// TwinCAT 3 PLC project TcoUrRobotics
// Title: TcoUrRobotics
// Company: Vortex.Library
// Author: TcOpenGroup
// ProjectVersion: 0.6.0.913
// ProgramVersion: 3.1.4024.12
// libraries:
//   Tc2_Standard, * (Beckhoff Automation GmbH)
//   Tc2_System, * (Beckhoff Automation GmbH)
//   Tc2_Utilities, * (Beckhoff Automation GmbH)
//   Tc3_Module, * (Beckhoff Automation GmbH)
//   TcoAbstractions, 0.6.0.913 (Vortex.Library)
//   TcoCore, 0.6.0.913 (Vortex.Library)
//   TcoIo, 0.6.0.913 (Vortex.Library)
//   TcoUtilities, 0.6.0.913 (Vortex.Library)
// project tree:
//   DUTs/ eTcoUrRoboticsRobotMode.TcDUT, TcoUrRoboticsInputData.TcDUT, TcoUrRoboticsOutputData.TcDUT, TcoUrRobotics_Config_v_1_x_x.TcDUT, TcoUrRobotics_Control_v_1_x_x.TcDUT, TcoUrRobotics_State_v_1_x_x.TcDUT, TcoUrRobotics_Status_v_1_x_x.TcDUT
//   DUTs/Input/ TcoUrRoboticsT2OBitRegs.TcDUT, TcoUrRoboticsT2OFloatRegs.TcDUT, TcoUrRoboticsT2ORobot.TcDUT, TcoUrRoboticsT2OIntRegs.TcDUT, TcoUrRoboticsT2OIo.TcDUT, TcoUrRoboticsT2OJoints.TcDUT, TcoUrRoboticsT2OSafety.TcDUT, TcoUrRoboticsT2OTcp.TcDUT, TcoUrRoboticsT2OTool.TcDUT
//   DUTs/Out/ TcoUrRobotics_O2TIo.TcDUT, TcoUrRobotics_O2TReg.TcDUT, TcoUrRobotics_O2TRobot.TcDUT
//   / PlcTask.TcTTO
//   POUs/ GetRobotModeDescription.TcPOU, MAIN.TcPOU
//   POUs/Prototypes/Cb3/IO/ TcoUrCb3_Inputs_v_3_x_x.TcDUT, TcoUrCb3_IO_v_3_x_x.TcDUT, TcoUrCb3_Outputs_v_3_x_x.TcDUT
//   POUs/Prototypes/Cb3/ TcoUrCb3_v_3_x_x.TcPOU
//   POUs/Prototypes/Eseries/IO/ TcoUrEseries_Inputs_v_5_x_x.TcDUT, TcoUrEseries_IO_v_5_x_x.TcDUT, TcoUrEseries_Outputs_v_5_x_x.TcDUT
//   POUs/Prototypes/Eseries/ TcoUrEseries_v_5_x_x.TcPOU
//   POUs/Prototypes/Generic/Inputs/ TcoUrRobotics_T2O_State_IO.TcDUT, TcoUrRobotics_T2O_IO_IO.TcDUT, TcoUrRobotics_T2O_Joints_IO.TcDUT, TcoUrRobotics_T2O_TCP_IO.TcDUT, TcoUrRobotics_T2O_BitRegs_IO.TcDUT, TcoUrRobotics_T2O_IntRegs_IO.TcDUT, TcoUrRobotics_T2O_FloatRegs_IO.TcDUT
//   POUs/Prototypes/Generic/Outputs/ TcoUrRobotics_O2T_Reg1_IO.TcDUT, TcoUrRobotics_O2T_Reg2_IO.TcDUT, TcoUrRobotics_O2T_Robot_IO.TcDUT
//   POUs/Prototypes/RoboticsTasks/Starts/ StartAtMainTask.TcPOU, StartMotorsAndProgramTask.TcPOU, StartMotorsProgramAndMovementsTask.TcPOU, StartMotorsTask.TcPOU, StartMovementsTask.TcPOU, StartProgramTask.TcPOU
//   POUs/Prototypes/RoboticsTasks/Stops/ StopMovementsAndProgramTask.TcPOU, StopMovementsTask.TcPOU, StopProgramTask.TcPOU
//   POUs/Prototypes/RoboticsTasks/ TcoUrRoboticsTask.TcPOU
// real-time tasks:
//   TASK PlcTask: cycle T#10ms, priority 20, ADS port 350
//   TASK PlcTask1: cycle T#10ms, priority 1, ADS port 351
//   TASK PN: cycle T#32ms, priority 2, ADS port 301
// I/O:
//   DEVICE Device 4 (EtherCAT) (disabled), AmsNetId 172.20.10.104.5.1
//     Term 1 (EK1100) [EK1100 EtherCAT Coupler (2A E-Bus)]
//       Term 2 (EL1008) [EL1008 8Ch. Dig. Input 24V, 3ms]
//       Term 3 (EL2008) [EL2008 8Ch. Dig. Output 24V, 0.5A]
//       Term 4 (EL3052) [EL3052 2Ch. Ana. Input 4-20mA]
//       Term 5 (EL9576) [EL9576 Brake chopper terminal]
//       Term 6 (EL7211-0010) [EL7211-0010 1Ch. MDP742 Servo motor output stage with OCT (50V, 4.5A RMS)]
//       Term 14 (EL7047) [EL7047 1Ch. Stepper motor output stage (50V, 5A)]
//       Term 8 (EL9011) [EL9011 End Terminal]
//   DEVICE Device 1 (EtherCAT) (disabled), AmsNetId 192.168.4.1.2.1
//     Drive 7 (IndraDrive MPB20) [IndraDrive MPB20]
//   DEVICE Device 2 (EtherCAT) (disabled), AmsNetId 192.168.4.1.3.1
//     Term 1 (EK1200) [EK1200-5000 EtherCAT Power supply (2A E-Bus)]
//       Term 10 (EK1122) [EK1122 2 port EtherCAT junction]
//       Term 13 (EL6631) [EL6631 PROFINET IO Controller]
//       Term 12 (EL1809) [EL1809 16Ch. Dig. Input 24V, 3ms]
//       Term 13 (EL2809) [EL2809 16Ch. Dig. Output 24V, 0.5A]
//       Term 15 (EL4004) [EL4004 4Ch. Ana. Output 0-10V, 12bit]
//       Term 16 (EL7342) [EL7342 2Ch. DC motor output stage (50V, 3.5A)]
//       Term 17 (EL4004) [EL4004 4Ch. Ana. Output 0-10V, 12bit]
//       Term 18 (EL6001) [EL6001 Interface (RS232)]
//       Term 10 (EL9011) [EL9011 End Terminal]
//   DEVICE Device 5 (Profinet Controller) (disabled), AmsNetId 192.168.4.1.6.1
//     ur-op-80r [Universal Robots A/S UR IO device, for PNIO controller with PDev 0000201]
//       modules: Term 1 (DAP Module), Term 3 (1_T2O State), Term 4 (2_T2O IO), Term 5 (3_T2O Joints), Term 6 (4_T2O TCP), Term 7 (5_T2O General Purpose Bit Registers), Term 8 (6_T2O General Purpose Int Registers), Term 9 (7_T2O General Purpose Float Registers), Term 10 (8_O2T Robot IO), Term 11 (9_O2T General Purpose Registers 1), Term 12 (10_O2T General Purpose Registers 2)
// variable links:
//   TcoUrRoboticsTests/TcoUrRoboticsTests Instance <-> Device 2 (EtherCAT)/Term 1 (EK1200)/Term 13 (EL2809)
//     PlcTask1 Outputs/GVL.A2[0] <-> Channel 1/Output
//     PlcTask1 Outputs/GVL.A2[1] <-> Channel 2/Output
//   TcoUrRoboticsTests/TcoUrRoboticsTests Instance <-> Device 5 (Profinet Controller)/ur-op-80r
//     PlcTask1 Inputs/GVL.Robot1.In.BitRegs.bArray <-> API/Term 7 (5_T2O General Purpose Bit Registers)/Subterm 9 (5_T2O General Purpose Bit Registers)/Inputs/T2O Bit Registers
//     PlcTask1 Inputs/GVL.Robot1.In.FloatRegs.bArray <-> API/Term 9 (7_T2O General Purpose Float Registers)/Subterm 11 (7_T2O General Purpose Float Registers)/Inputs/T2O Float Registers
//     PlcTask1 Inputs/GVL.Robot1.In.IO.bArray <-> API/Term 4 (2_T2O IO)/Subterm 6 (2_T2O IO)/Inputs/T2O IO
//     PlcTask1 Inputs/GVL.Robot1.In.IntRegs.bArray <-> API/Term 8 (6_T2O General Purpose Int Registers)/Subterm 10 (6_T2O General Purpose Int Registers)/Inputs/T2O Int Registers
//     PlcTask1 Inputs/GVL.Robot1.In.Joints.bArray <-> API/Term 5 (3_T2O Joints)/Subterm 7 (3_T2O Joints)/Inputs/T2O Joints
//     PlcTask1 Inputs/GVL.Robot1.In.State.bArray <-> API/Term 3 (1_T2O State)/Subterm 5 (1_T2O State)/Inputs/T2O State
//     PlcTask1 Inputs/GVL.Robot1.In.TCP.bArray <-> API/Term 6 (4_T2O TCP)/Subterm 8 (4_T2O TCP)/Inputs/T2O TCP
//     PlcTask1 Inputs/GVL.Robot1.PnIoBoxDiag <-> Inputs/PnIoBoxDiag
//     PlcTask1 Inputs/GVL.Robot1.PnIoBoxState <-> Inputs/PnIoBoxState
//     PlcTask1 Outputs/GVL.Robot1.Out.Reg1.bArray <-> API/Term 11 (9_O2T General Purpose Registers 1)/Subterm 13 (9_O2T General Purpose Registers 1)/Outputs/O2T Reg 1
//     PlcTask1 Outputs/GVL.Robot1.Out.Reg2.bArray <-> API/Term 12 (10_O2T General Purpose Registers 2)/Subterm 14 (10_O2T General Purpose Registers 2)/Outputs/O2T Reg 2
//     PlcTask1 Outputs/GVL.Robot1.Out.RobotIO.bArray <-> API/Term 10 (8_O2T Robot IO)/Subterm 12 (8_O2T Robot IO)/Outputs/O2T IO

CONFIGURATION TcoUrRobotics
    RESOURCE PLC ON TwinCAT3
        TASK PlcTask(INTERVAL := T#10ms, PRIORITY := 20);
        PROGRAM MAIN WITH PlcTask : MAIN;
    END_RESOURCE
END_CONFIGURATION

// ---- DUTs/eTcoUrRoboticsRobotMode.TcDUT
{attribute 'qualified_only'}
{attribute 'strict'}
TYPE eTcoUrRoboticsRobotMode :
(
    DISCONNECTED := 0,
    SAFETY := 1,
    BOOTING := 2,
    POWER_OFF := 3,
    POWER_ON := 4,
    IDLE := 5,
    BACKDRIVE := 6,
    RUNNING := 7,
    UPDATING_FIRMWARE := 8
);
END_TYPE

// ---- DUTs/Input/TcoUrRoboticsT2OBitRegs.TcDUT
TYPE TcoUrRoboticsT2OBitRegs :
STRUCT
    {attribute addProperty Name "<#Bit registers#>"}
    Register : ARRAY[0..63] OF BOOL;
END_STRUCT
END_TYPE

// ---- DUTs/Input/TcoUrRoboticsT2OFloatRegs.TcDUT
TYPE TcoUrRoboticsT2OFloatRegs :
STRUCT
    {attribute addProperty Name "<#Float registers#>"}
    Register : ARRAY[0..23] OF REAL;
END_STRUCT
END_TYPE

// ---- DUTs/Input/TcoUrRoboticsT2ORobot.TcDUT
TYPE TcoUrRoboticsT2ORobot :
STRUCT
    {attribute addProperty Name "<#Controller major version#>"}
    ControllerMajorVersion : USINT;
    {attribute addProperty Name "<#Controller minor version#>"}
    ControllerMinorVersion : USINT;
    {attribute addProperty Name "<#Reserved#>"}
    Reserved : UINT;
    {attribute addProperty Name "<#Robot mode#>"}
    RobotMode : USINT;
    {attribute addProperty Name "<#Real time machine seconds#>"}
    RealtimeMachineSeconds : USINT;
    {attribute addProperty Name "<#Real time machine milliseconds#>"}
    RealtimeMachineMilliseconds : UINT;
    {attribute addProperty Name "<#Real time machine minutes#>"}
    RealtimeMachineMinutes : USINT;
    {attribute addProperty Name "<#Real time machine hours#>"}
    RealtimeMachineHours : USINT;
    {attribute addProperty Name "<#Real time machine days#>"}
    RealtimeMachineDays : UINT;
    {attribute addProperty Name "<#Robot current [A]#>"}
    RobotCurrent : REAL;
    {attribute addProperty Name "<#PW: Is power on#>"}
    PW_IsPowerOn : BOOL;
    {attribute addProperty Name "<#PR: Is program running#>"}
    PR_IsProgramRunning : BOOL;
    {attribute addProperty Name "<#TB: Is teach button pressed#>"}
    TB_IsTeachButtonPressed : BOOL;
    {attribute addProperty Name "<#PB: Is power button pressed#>"}
    PB_IsPowerButtonPressed : BOOL;
    {attribute addProperty Name "<#Speed slider fraction#>"}
    SpeedSliderFraction : REAL;
END_STRUCT
END_TYPE

// ---- DUTs/Input/TcoUrRoboticsT2OIntRegs.TcDUT
TYPE TcoUrRoboticsT2OIntRegs :
STRUCT
    {attribute addProperty Name "<#Int registers#>"}
    Register : ARRAY[0..23] OF DINT;
END_STRUCT
END_TYPE

// ---- DUTs/Input/TcoUrRoboticsT2OIo.TcDUT
TYPE TcoUrRoboticsT2OIo :
STRUCT
    {attribute addProperty Name "<#Standard digital inputs#>"}
    StandardDigitalInputs : USINT;
    {attribute addProperty Name "<#Configurable digital inputs#>"}
    ConfigurableDigitalInputs : USINT;
    {attribute addProperty Name "<#Standard digital outputs#>"}
    StandardDigitalOutputs : USINT;
    {attribute addProperty Name "<#Configurable digital outputs#>"}
    ConfigurableDigitalOutputs : USINT;
    {attribute addProperty Name "<#Analog I/O types#>"}
    AnalogIoTypes : USINT;
    {attribute addProperty Name "<#Standard analog input [A or V]#>"}
    StandardAnalogInput : ARRAY[0..1] OF REAL;
    {attribute addProperty Name "<#Standard analog output [A or V]#>"}
    StandardAnalogOutput : ARRAY[0..1] OF REAL;
    {attribute addProperty Name "<#I/O current [A]#>"}
    Current : REAL;
    {attribute addProperty Name "<#Euromap67 input bits#>"}
    Euromap67InputBits : ARRAY[0..31] OF BOOL;
    {attribute addProperty Name "<#Euromap67 output bits#>"}
    Euromap67OutputBits : ARRAY[0..31] OF BOOL;
    {attribute addProperty Name "<#Euromap67 24V voltage#>"}
    Euromap6724Voltage : REAL;
    {attribute addProperty Name "<#Euromap67 24V current#>"}
    Euromap6724VCurrent : REAL;
END_STRUCT
END_TYPE

// ---- DUTs/Input/TcoUrRoboticsT2OJoints.TcDUT
TYPE TcoUrRoboticsT2OJoints :
STRUCT
    {attribute addProperty Name "<#Joint position [rad]#>"}
    JointPosition : ARRAY[0..5] OF REAL;
    {attribute addProperty Name "<#Joint velocity [rad/s]#>"}
    JointVelocity : ARRAY[0..5] OF REAL;
    {attribute addProperty Name "<#Joint current [A]#>"}
    JointCurrent : ARRAY[0..5] OF REAL;
    {attribute addProperty Name "<#Joint temperature [°C]#>"}
    JointTemperature : ARRAY[0..5] OF REAL;
    {attribute addProperty Name "<#Joint mode#>"}
    JointMode : ARRAY[0..5] OF USINT;
END_STRUCT
END_TYPE

// ---- DUTs/Input/TcoUrRoboticsT2OSafety.TcDUT
TYPE TcoUrRoboticsT2OSafety :
STRUCT
    {attribute addProperty Name "<#Safety mode#>"}
    SafetyMode : USINT;
    {attribute addProperty Name "<#NO: Is normal mode#>"}
    NO_IsNormalMode : BOOL;
    {attribute addProperty Name "<#RD: Is reduced mode#>"}
    RD_IsReducedMode : BOOL;
    {attribute addProperty Name "<#PS: Is protective stopped#>"}
    PS_IsProtectiveStopped : BOOL;
    {attribute addProperty Name "<#RC: Is recovery mode#>"}
    RC_IsRecoveryMode : BOOL;
    {attribute addProperty Name "<#SS: Is safeguard stopped#>"}
    SS_IsSafeguardStopped : BOOL;
    {attribute addProperty Name "<#SES: Is system emergency stopped#>"}
    SES_IsSystemEmergencyStopped : BOOL;
    {attribute addProperty Name "<#RES: Is robot emergency stopped#>"}
    RES_IsRobotEmergencyStopped : BOOL;
    {attribute addProperty Name "<#ES: Is emergency stopped#>"}
    ES_IsEmergencyStopped : BOOL;
    {attribute addProperty Name "<#VL: Is violation#>"}
    VL_IsViolation : BOOL;
    {attribute addProperty Name "<#FT: Is fault#>"}
    FT_IsFault : BOOL;
    {attribute addProperty Name "<#ST: Is stopped due TO safety#>"}
    ST_IsStoppedDueSafety : BOOL;
END_STRUCT
END_TYPE

// ---- DUTs/Input/TcoUrRoboticsT2OTcp.TcDUT
TYPE TcoUrRoboticsT2OTcp :
STRUCT
    {attribute addProperty Name "<#Actual TCP Position#>"}
    Postition : TcoAbstractions.TcoRoboticsCoordinates;
    {attribute addProperty Name "<#Actual TCP Velocity#>"}
    Velocity : TcoAbstractions.TcoRoboticsCoordinates;
    {attribute addProperty Name "<#Actual TCP Force#>"}
    Force : TcoAbstractions.TcoRoboticsBasicCoordinates;
    {attribute addProperty Name "<#Actual TCP Torque#>"}
    Torque : TcoAbstractions.TcoRoboticsBasicCoordinates;
    {attribute addProperty Name "<#TCP force scalar [N]#>"}
    TCP_ForceScalar : REAL;
END_STRUCT
END_TYPE

// ---- DUTs/Input/TcoUrRoboticsT2OTool.TcDUT
TYPE TcoUrRoboticsT2OTool :
STRUCT
    {attribute addProperty Name "<#Tool mode#>"}
    ToolMode : USINT;
    {attribute addProperty Name "<#TDI: Tool Digital Inputs#>"}
    TDI_ToolDigitalInputs : USINT;
    {attribute addProperty Name "<#TDO: Tool Digital Outputs#>"}
    TDO_ToolDigitalOutputs : USINT;
    {attribute addProperty Name "<#TAIT: Tool Analog Input Types#>"}
    TAIT_ToolAnalogInputTypes : USINT;
    {attribute addProperty Name "<#Tool analog input [A OR V]#>"}
    ToolAnalogInput : ARRAY[0..1] OF REAL;
    {attribute addProperty Name "<#Tool output voltage [V]#>"}
    ToolOutputVoltage : REAL;
    {attribute addProperty Name "<#Tool current [A]#>"}
    ToolCurrent : REAL;
END_STRUCT
END_TYPE

// ---- DUTs/Out/TcoUrRobotics_O2TIo.TcDUT
TYPE TcoUrRobotics_O2TIo :
STRUCT
    {attribute addProperty Name "<#Standard digital output mask#>"}
    StandardDigitalOutputMask : USINT;
    {attribute addProperty Name "<#Configurable digital output mask#>"}
    ConfigurableDigitalOutputMask : USINT;
    {attribute addProperty Name "<#Standard digital outputs#>"}
    StandardDigitalOutputs : USINT;
    {attribute addProperty Name "<#Configurable digital outputs#>"}
    ConfigurableDdigitalOutputs : USINT;
    {attribute addProperty Name "<#AOM: Analog output mask#>"}
    AOM_AnalogOutputMask : USINT;
    {attribute addProperty Name "<#AOT: Analog output types#>"}
    AOT_AnalogOutputTypes : USINT;
    {attribute addProperty Name "<#TDOM: Tool digital output mask#>"}
    TDOM_ToolDigitalOutputMask : USINT;
    {attribute addProperty Name "<#TDO: Tool digital output#>"}
    TDO_ToolDigitalOutput : USINT;
    {attribute addProperty Name "<#Standard analog output#>"}
    StandardAnalogOutput : ARRAY[0..1] OF REAL;
END_STRUCT
END_TYPE

// ---- DUTs/Out/TcoUrRobotics_O2TReg.TcDUT
TYPE TcoUrRobotics_O2TReg :
STRUCT
    {attribute addProperty Name "<#Bit registers#>"}
    Bits : ARRAY[0..31] OF BOOL;
    {attribute addProperty Name "<#Int registers#>"}
    Ints : ARRAY[0..11] OF DINT;
    {attribute addProperty Name "<#Float registers#>"}
    Floats : ARRAY[0..11] OF REAL;
END_STRUCT
END_TYPE

// ---- DUTs/Out/TcoUrRobotics_O2TRobot.TcDUT
TYPE TcoUrRobotics_O2TRobot :
STRUCT
    {attribute addProperty Name "<#SSM: Speed slider fraction mask#>"}
    SSM_SpeedSliderFractionMask : BOOL;
    {attribute addProperty Name "<#Speed slider fraction#>"}
    SpeedSliderFraction : REAL;
END_STRUCT
END_TYPE

// ---- DUTs/TcoUrRoboticsInputData.TcDUT
TYPE TcoUrRoboticsInputData :
STRUCT
    {attribute addProperty Name "<#Robot#>"}
    Robot : TcoUrRoboticsT2ORobot;
    {attribute addProperty Name "<#State#>"}
    Safety : TcoUrRoboticsT2OSafety;
    {attribute addProperty Name "<#IO state#>"}
    IO : TcoUrRoboticsT2OIo;
    {attribute addProperty Name "<#Tool state#>"}
    Tool : TcoUrRoboticsT2OTool;
    {attribute addProperty Name "<#Joints#>"}
    Joints : TcoUrRoboticsT2OJoints;
    {attribute addProperty Name "<#TCP#>"}
    TCP : TcoUrRoboticsT2OTcp;
    {attribute addProperty Name "<#Bits#>"}
    Bits : TcoUrRoboticsT2OBitRegs;
    {attribute addProperty Name "<#Ints#>"}
    Ints : TcoUrRoboticsT2OIntRegs;
    {attribute addProperty Name "<#Floats#>"}
    Floats : TcoUrRoboticsT2OFloatRegs;
END_STRUCT
END_TYPE

// ---- DUTs/TcoUrRoboticsOutputData.TcDUT
TYPE TcoUrRoboticsOutputData :
STRUCT
    {attribute addProperty Name "<#Speed#>"}
    Speed : TcoUrRobotics_O2TRobot;
    {attribute addProperty Name "<#IO#>"}
    IO : TcoUrRobotics_O2TIo;
    {attribute addProperty Name "<#Reg 1#>"}
    Reg1 : TcoUrRobotics_O2TReg;
    {attribute addProperty Name "<#Reg 2#>"}
    Reg2 : TcoUrRobotics_O2TReg;
END_STRUCT
END_TYPE

// ---- DUTs/TcoUrRobotics_Config_v_1_x_x.TcDUT
TYPE TcoUrRobotics_Config_v_1_x_x :
STRUCT
    InfoTime : TIME := T#2S;
    ErrorTime : TIME := T#0S;
    RemotePowerOnEnabled : BOOL := FALSE;
    RemotePowerOnPulse : TIME := T#500MS;
    IpAddress : STRING;
END_STRUCT
END_TYPE

// ---- DUTs/TcoUrRobotics_Control_v_1_x_x.TcDUT
TYPE TcoUrRobotics_Control_v_1_x_x :
STRUCT
    {attribute addProperty Name "<#Start program#>"}
    Start : BOOL;
    {attribute addProperty Name "<#Stop program#>"}
    Stop : BOOL;
    {attribute addProperty Name "<#Pause program#>"}
    Pause : BOOL;
    {attribute addProperty Name "<#Set motor on#>"}
    MotorOn : BOOL;
    {attribute addProperty Name "<#Run action#>"}
    RunAction : BOOL;
    {attribute addProperty Name "<#Master mode#>"}
    MasterMode : BYTE;
    {attribute addProperty Name "<#Tool 1 retract#>"}
    Tool_1_Retract : BOOL;
    {attribute addProperty Name "<#Tool 1 extend#>"}
    Tool_1_Extend : BOOL;
    {attribute addProperty Name "<#Tool 2 retract#>"}
    Tool_2_Retract : BOOL;
    {attribute addProperty Name "<#Tool 2 extend#>"}
    Tool_2_Extend : BOOL;
    {attribute addProperty Name "<#Tool 3 retract#>"}
    Tool_3_Retract : BOOL;
    {attribute addProperty Name "<#Tool 3 extend#>"}
    Tool_3_Extend : BOOL;
    {attribute addProperty Name "<#Tool 4 retract#>"}
    Tool_4_Retract : BOOL;
    {attribute addProperty Name "<#Tool 4 extend#>"}
    Tool_4_Extend : BOOL;
    {attribute addProperty Name "<#Zones#>"}
    Zone : DINT;
    {attribute addProperty Name "<#In position#>"}
    InPosition : DINT;
    {attribute addProperty Name "<#Action number#>"}
    ActionNo : DINT;
    {attribute addProperty Name "<#Global robot speed#>"}
    GlobalSpeed : DINT;
    {attribute addProperty Name "<#Tool number#>"}
    ToolNo : DINT;
    {attribute addProperty Name "<#Workobject number#>"}
    WorkobjectNo : DINT;
    {attribute addProperty Name "<#Point number#>"}
    PointNo : DINT;
    {attribute addProperty Name "<#User specific speed 1#>"}
    UserSpecSpeed1 : REAL;
    {attribute addProperty Name "<#User specific speed 2#>"}
    UserSpecSpeed2 : REAL;
    {attribute  addProperty Name "<#Coordinates#>"}
    Coordinates : TcoAbstractions.TcoRoboticsCoordinates;
    {attribute addProperty Name "<UR Specific#>"}
    Outputs : TcoUrRoboticsOutputData;
END_STRUCT
END_TYPE

// ---- DUTs/TcoUrRobotics_State_v_1_x_x.TcDUT
TYPE TcoUrRobotics_State_v_1_x_x :
STRUCT
    {attribute addProperty Name "<#Robot Mode#>"}
    RobotMode : eTcoUrRoboticsRobotMode;
    {attribute addProperty Name "<#In area 1#>"}
    InArea_1 : BOOL;
    {attribute addProperty Name "<#In area 2#>"}
    InArea_2 : BOOL;
    {attribute addProperty Name "<#In area 3#>"}
    InArea_3 : BOOL;
    {attribute addProperty Name "<#In area 4#>"}
    InArea_4 : BOOL;
    {attribute addProperty Name "<#In position 1#>"}
    InPosition_1 : BOOL;
    {attribute addProperty Name "<#In position 2#>"}
    InPosition_2 : BOOL;
    {attribute addProperty Name "<#In position 3#>"}
    InPosition_3 : BOOL;
    {attribute addProperty Name "<#In position 4#>"}
    InPosition_4 : BOOL;
    {attribute addProperty Name "<#Zones#>"}
    Zone : DINT;
    {attribute addProperty Name "<#In position#>"}
    InPosition : DINT;
    {attribute addProperty Name "<#Tool 1 retract#>"}
    Tool_1_Retract : BOOL;
    {attribute addProperty Name "<#Tool 1 extend#>"}
    Tool_1_Extend : BOOL;
    {attribute addProperty Name "<#Tool 2 retract#>"}
    Tool_2_Retract : BOOL;
    {attribute addProperty Name "<#Tool 2 extend#>"}
    Tool_2_Extend : BOOL;
    {attribute addProperty Name "<#Tool 3 retract#>"}
    Tool_3_Retract : BOOL;
    {attribute addProperty Name "<#Tool 3 extend#>"}
    Tool_3_Extend : BOOL;
    {attribute addProperty Name "<#Tool 4 retract#>"}
    Tool_4_Retract : BOOL;
    {attribute addProperty Name "<#Tool 4 extend#>"}
    Tool_4_Extend : BOOL;
    {attribute addProperty Name "<#Action number#>"}
    ActionNo : DINT;
    {attribute addProperty Name "<#Global speed#>"}
    GlobalSpeed : DINT;
    {attribute addProperty Name "<#Tool number#>"}
    ToolNo : DINT;
    {attribute addProperty Name "<#Workobject number#>"}
    WorkobjectNo : DINT;
    {attribute addProperty Name "<#PointNumber#>"}
    PointNo : DINT;
    {attribute addProperty Name "<#User specific speed 1#>"}
    UserSpecSpeed1 : REAL;
    {attribute addProperty Name "<#User specific speed 2#>"}
    UserSpecSpeed2 : REAL;
    {attribute  addProperty Name "<#Coordinates#>"}
    Coordinates : TcoAbstractions.TcoRoboticsCoordinates;
    {attribute  addProperty Name "<#UR Specific#>"}
    Inputs : TcoUrRoboticsInputData;
END_STRUCT
END_TYPE

// ---- DUTs/TcoUrRobotics_Status_v_1_x_x.TcDUT
TYPE TcoUrRobotics_Status_v_1_x_x :
STRUCT
    ActionDescription : STRING(100);
    State : TcoUrRobotics_State_v_1_x_x;
END_STRUCT
END_TYPE

// ---- POUs/Prototypes/Cb3/IO/TcoUrCb3_Inputs_v_3_x_x.TcDUT
TYPE TcoUrCb3_Inputs_v_3_x_x :
STRUCT
    {attribute addProperty Name "<#State#>"}
    State : TcoUrRobotics_T2O_State_IO;
    {attribute addProperty Name "<#IO#>"}
    IO : TcoUrRobotics_T2O_IO_IO;
    {attribute addProperty Name "<#Joints#>"}
    Joints : TcoUrRobotics_T2O_Joints_IO;
    {attribute addProperty Name "<#TCP#>"}
    TCP : TcoUrRobotics_T2O_TCP_IO;
    {attribute addProperty Name "<#Bit registers#>"}
    BitRegs : TcoUrRobotics_T2O_BitRegs_IO;
    {attribute addProperty Name "<#Int registers#>"}
    IntRegs : TcoUrRobotics_T2O_IntRegs_IO;
    {attribute addProperty Name "<#Float registers#>"}
    FloatRegs : TcoUrRobotics_T2O_FloatRegs_IO;
END_STRUCT
END_TYPE

// ---- POUs/Prototypes/Cb3/IO/TcoUrCb3_IO_v_3_x_x.TcDUT
TYPE TcoUrCb3_IO_v_3_x_x :
STRUCT
    PnIoBoxState AT %I* : UINT;
    PnIoBoxDiag AT %I* : UINT;
    PnIoBoxCtrl AT %Q* : UINT;
    {attribute addProperty Name "<#IN#>"}
    In : TcoUrCb3_Inputs_v_3_x_x;
    {attribute addProperty Name "<#OUT#>"}
    Out : TcoUrCb3_Outputs_v_3_x_x;
END_STRUCT
END_TYPE

// ---- POUs/Prototypes/Cb3/IO/TcoUrCb3_Outputs_v_3_x_x.TcDUT
TYPE TcoUrCb3_Outputs_v_3_x_x :
STRUCT
    {attribute addProperty Name "<#RobotIO#>"}
    RobotIO : TcoUrRobotics_O2T_Robot_IO;
    {attribute addProperty Name "<#Reg2#>"}
    Reg1 : TcoUrRobotics_O2T_Reg1_IO;
    {attribute addProperty Name "<#Reg2#>"}
    Reg2 : TcoUrRobotics_O2T_Reg2_IO;
END_STRUCT
END_TYPE

// ---- POUs/Prototypes/Eseries/IO/TcoUrEseries_Inputs_v_5_x_x.TcDUT
TYPE TcoUrEseries_Inputs_v_5_x_x :
STRUCT
    {attribute addProperty Name "<#State#>"}
    State : TcoUrRobotics_T2O_State_IO;
    {attribute addProperty Name "<#IO#>"}
    IO : TcoUrRobotics_T2O_IO_IO;
    {attribute addProperty Name "<#Joints#>"}
    Joints : TcoUrRobotics_T2O_Joints_IO;
    {attribute addProperty Name "<#TCP#>"}
    TCP : TcoUrRobotics_T2O_TCP_IO;
    {attribute addProperty Name "<#Bit registers#>"}
    BitRegs : TcoUrRobotics_T2O_BitRegs_IO;
    {attribute addProperty Name "<#Int registers#>"}
    IntRegs : TcoUrRobotics_T2O_IntRegs_IO;
    {attribute addProperty Name "<#Float registers#>"}
    FloatRegs : TcoUrRobotics_T2O_FloatRegs_IO;
END_STRUCT
END_TYPE

// ---- POUs/Prototypes/Eseries/IO/TcoUrEseries_IO_v_5_x_x.TcDUT
TYPE TcoUrEseries_IO_v_5_x_x :
STRUCT
    PnIoBoxState AT %I* : UINT;
    PnIoBoxDiag AT %I* : UINT;
    PnIoBoxCtrl AT %Q* : UINT;
    {attribute addProperty Name "<#IN#>"}
    In : TcoUrEseries_Inputs_v_5_x_x;
    {attribute addProperty Name "<#OUT#>"}
    Out : TcoUrEseries_Outputs_v_5_x_x;
END_STRUCT
END_TYPE

// ---- POUs/Prototypes/Eseries/IO/TcoUrEseries_Outputs_v_5_x_x.TcDUT
TYPE TcoUrEseries_Outputs_v_5_x_x :
STRUCT
    {attribute addProperty Name "<#RobotIO#>"}
    RobotIO : TcoUrRobotics_O2T_Robot_IO;
    {attribute addProperty Name "<#Reg2#>"}
    Reg1 : TcoUrRobotics_O2T_Reg1_IO;
    {attribute addProperty Name "<#Reg2#>"}
    Reg2 : TcoUrRobotics_O2T_Reg2_IO;
END_STRUCT
END_TYPE

// ---- POUs/Prototypes/Generic/Inputs/TcoUrRobotics_T2O_State_IO.TcDUT
TYPE TcoUrRobotics_T2O_State_IO :
STRUCT
    bArray AT %I* : ARRAY[0..31] OF BYTE;
END_STRUCT
END_TYPE

// ---- POUs/Prototypes/Generic/Inputs/TcoUrRobotics_T2O_IO_IO.TcDUT
TYPE TcoUrRobotics_T2O_IO_IO :
STRUCT
    bArray AT %I* : ARRAY[0..67] OF BYTE;
END_STRUCT
END_TYPE

// ---- POUs/Prototypes/Generic/Inputs/TcoUrRobotics_T2O_Joints_IO.TcDUT
TYPE TcoUrRobotics_T2O_Joints_IO :
STRUCT
    bArray AT %I* : ARRAY[0..103] OF BYTE;
END_STRUCT
END_TYPE

// ---- POUs/Prototypes/Generic/Inputs/TcoUrRobotics_T2O_TCP_IO.TcDUT
TYPE TcoUrRobotics_T2O_TCP_IO :
STRUCT
    bArray AT %I* : ARRAY[0..75] OF BYTE;
END_STRUCT
END_TYPE

// ---- POUs/Prototypes/Generic/Inputs/TcoUrRobotics_T2O_BitRegs_IO.TcDUT
TYPE TcoUrRobotics_T2O_BitRegs_IO :
STRUCT
    bArray AT %I* : ARRAY[0..7] OF BYTE;
END_STRUCT
END_TYPE

// ---- POUs/Prototypes/Generic/Inputs/TcoUrRobotics_T2O_IntRegs_IO.TcDUT
TYPE TcoUrRobotics_T2O_IntRegs_IO :
STRUCT
    bArray AT %I* : ARRAY[0..95] OF BYTE;
END_STRUCT
END_TYPE

// ---- POUs/Prototypes/Generic/Inputs/TcoUrRobotics_T2O_FloatRegs_IO.TcDUT
TYPE TcoUrRobotics_T2O_FloatRegs_IO :
STRUCT
    bArray AT %I* : ARRAY[0..95] OF BYTE;
END_STRUCT
END_TYPE

// ---- POUs/Prototypes/Generic/Outputs/TcoUrRobotics_O2T_Reg1_IO.TcDUT
TYPE TcoUrRobotics_O2T_Reg1_IO :
STRUCT
    bArray AT %Q* : ARRAY[0..99] OF BYTE;
END_STRUCT
END_TYPE

// ---- POUs/Prototypes/Generic/Outputs/TcoUrRobotics_O2T_Reg2_IO.TcDUT
TYPE TcoUrRobotics_O2T_Reg2_IO :
STRUCT
    bArray AT %Q* : ARRAY[0..99] OF BYTE;
END_STRUCT
END_TYPE

// ---- POUs/Prototypes/Generic/Outputs/TcoUrRobotics_O2T_Robot_IO.TcDUT
TYPE TcoUrRobotics_O2T_Robot_IO :
STRUCT
    bArray AT %Q* : ARRAY[0..23] OF BYTE;
END_STRUCT
END_TYPE

// ---- POUs/MAIN.TcPOU
PROGRAM MAIN
VAR
END_VAR

END_PROGRAM

// ---- POUs/GetRobotModeDescription.TcPOU
FUNCTION GetRobotModeDescription : eTcoUrRoboticsRobotMode
VAR_INPUT
    inMode : USINT;
END_VAR
VAR
    retVal : eTcoUrRoboticsRobotMode;
END_VAR

CASE inMode OF
    0:
        retVal := eTcoUrRoboticsRobotMode.DISCONNECTED;
    1:
        retVal := eTcoUrRoboticsRobotMode.SAFETY;
    2:
        retVal := eTcoUrRoboticsRobotMode.BOOTING;
    3:
        retVal := eTcoUrRoboticsRobotMode.POWER_OFF;
    4:
        retVal := eTcoUrRoboticsRobotMode.POWER_ON;
    5:
        retVal := eTcoUrRoboticsRobotMode.IDLE;
    6:
        retVal := eTcoUrRoboticsRobotMode.BACKDRIVE;
    7:
        retVal := eTcoUrRoboticsRobotMode.RUNNING;
    8:
        retVal := eTcoUrRoboticsRobotMode.UPDATING_FIRMWARE;
END_CASE

GetRobotModeDescription := retVal;

END_FUNCTION

// ---- POUs/Prototypes/Cb3/TcoUrCb3_v_3_x_x.TcPOU
FUNCTION_BLOCK TcoUrCb3_v_3_x_x EXTENDS TcoIo.TcoPnIoComponent IMPLEMENTS TcoAbstractions.ITcoRobotics
VAR_IN_OUT
    inoData : TcoUrCb3_IO_v_3_x_x;
    inoPowerOnPulse : BOOL;
END_VAR
VAR
    {attribute addProperty Name "<#Status#>"}
    {attribute clr [ReadOnly()]}
    _status : TcoUrRobotics_Status_v_1_x_x;
    {attribute addProperty Name "<#Control#>"}
    _control : TcoUrRobotics_Control_v_1_x_x;
    {attribute addProperty Name "<#Config#>"}
    _config : TcoUrRobotics_Config_v_1_x_x;
    {attribute addProperty Name "<#PN Error#>"}
    {attribute clr [ReadOnly()]}
    _pnError : BOOL;
    _someTaskIsActive : BOOL;
    _stopTasksAreActive : BOOL;
END_VAR
VAR
    {attribute addProperty Name "<#Start at Main#>"}
    _startAtMainTask : StartAtMainTask(THIS^);
    {attribute addProperty Name "<#Start motors and program#>"}
    _startMotorsAndProgramTask : StartMotorsAndProgramTask(THIS^);
    {attribute addProperty Name "<#Start program#>"}
    _startProgramTask : StartProgramTask(THIS^);
    {attribute addProperty Name "<#Start motors#>"}
    _startMotorsTask : StartMotorsTask(THIS^);
    {attribute addProperty Name "<#Start movements#>"}
    _startMovementsTask : StartMovementsTask(THIS^);
    {attribute addProperty Name "<#Start motors program and movements#>"}
    _startMotorsProgramAndMovementsTask : StartMotorsProgramAndMovementsTask(THIS^);
    {attribute addProperty Name "<#Stop movements#>"}
    _stopMovementsTask : StopMovementsTask(THIS^);
    {attribute addProperty Name "<#Stop movenents and program#>"}
    _stopMovementsAndProgramTask : StopMovementsAndProgramTask(THIS^);
    {attribute addProperty Name "<#Stop program#>"}
    _stopProgramTask : StopProgramTask(THIS^);
    {attribute addProperty Name "<#Power On Task#>"}
    _powerOnTask : TcoCore.TcoTask(THIS^);
    {attribute addProperty Name "<#Restore#>"}
    _restoreTask : TcoCore.TcoTask(THIS^);
END_VAR
VAR
    {attribute 'hide'}
    _sb : TcoCore.StringBuilder;
END_VAR

IF NOT __ISVALIDREF(inoData) THEN
    Messenger.Post('Invalid reference', TcoCore.eMessageCategory.ProgrammingError);
    RETURN;
END_IF

SUPER^(inPnIoBoxState := THIS^.inoData.PnIoBoxState, inPnIoBoxDiag := THIS^.inoData.PnIoBoxDiag);
_pnError := not _profinetReady;
UpdateStatus();
_stopTasksAreActive := _stopMovementsTask.Busy AND _stopMovementsAndProgramTask.Busy AND _stopProgramTask.Busy;
_startAtMainTask.Enabled := NOT _stopTasksAreActive;
_startAtMainTask(inoConfig := _config, inoControl := _control, inoStatus := _status);
_startProgramTask.Enabled := NOT _stopTasksAreActive;
_startProgramTask(inoConfig := _config, inoControl := _control, inoStatus := _status);
_startMotorsTask.Enabled := NOT _stopTasksAreActive AND NOT _startMotorsProgramAndMovementsTask.Busy AND NOT _startMotorsAndProgramTask.Busy;
_startMotorsTask(inoConfig := _config, inoControl := _control, inoStatus := _status);
_startMotorsAndProgramTask.Enabled := NOT _stopTasksAreActive AND NOT _startProgramTask.Busy AND NOT _startMotorsTask.Busy;
_startMotorsAndProgramTask(inoConfig := _config, inoControl := _control, inoStatus := _status);
_startMovementsTask.Enabled := NOT _startMotorsProgramAndMovementsTask.Busy;
_startMovementsTask(inoConfig := _config, inoControl := _control, inoStatus := _status);
_startMotorsProgramAndMovementsTask.Enabled := NOT _startMovementsTask.Busy;

_startMotorsProgramAndMovementsTask(refStartMotorsAndProgramTask := _startMotorsAndProgramTask,
    inoConfig := _config,
    inoControl := _control,
    inoStatus := _status);

_stopMovementsTask.Enabled := TRUE;
_stopMovementsTask(inoConfig := _config, inoControl := _control, inoStatus := _status);
_stopProgramTask.Enabled := TRUE;
_stopProgramTask(inoConfig := _config, inoControl := _control, inoStatus := _status);
_stopMovementsAndProgramTask.Enabled := NOT _stopProgramTask.Busy AND NOT _stopProgramTask.Busy;
_stopMovementsAndProgramTask(inoConfig := _config, inoControl := _control, inoStatus := _status);
//*************POWER ON********************
_powerOnTask.Enabled := _status.State.RobotMode = eTcoUrRoboticsRobotMode.DISCONNECTED AND _config.RemotePowerOnEnabled;

IF _powerOnTask.Execute() THEN
    inoPowerOnPulse := TRUE;
    Messenger.Notify('<#POWER ON PULSE WAS SEND TO CONTROLER#>');
    _powerOnTask.DoneWhen(_powerOnTask.ElapsedTime > _config.RemotePowerOnPulse);
END_IF

IF inoPowerOnPulse AND _powerOnTask.Done OR NOT _config.RemotePowerOnEnabled THEN
    inoPowerOnPulse := FALSE;
END_IF
//****************************************
//*************RESTORE********************
_restoreTask.Enabled := TRUE;

IF _restoreTask.Execute() THEN
    Restore();
    _restoreTask.DoneWhen(TRUE);
END_IF

//****************************************
_someTaskIsActive := _startAtMainTask.Busy OR
    _startMotorsAndProgramTask.Busy OR
    _startMovementsTask.Busy OR
    _startMovementsTask.Busy OR
    _stopMovementsTask.Busy OR
    _stopMovementsAndProgramTask.Busy OR
    _stopProgramTask.Busy;

//do not publish diagnostic message when component is not used
IF _someTaskIsActive THEN
    IF (_status.State.Inputs.Safety.ES_IsEmergencyStopped) THEN
        Messenger.Error('<#Emergency stop active#>');
    END_IF;

    IF (_status.State.Inputs.Safety.ST_IsStoppedDueSafety) THEN
        Messenger.Warning('<#Stopped due safety#>');
    END_IF;
END_IF;

UpdateControl();

(*~
    <docu>
        <summary>
            Gets the configuration of the IRC 5.
        </summary>
    </docu>
~*)
PROPERTY Config : REFERENCE TO TcoUrRobotics_Config_v_1_x_x
GET
Config REF= _config;
END_GET
END_PROPERTY

PROPERTY PUBLIC Control : REFERENCE TO TcoUrRobotics_Control_v_1_x_x
GET
Control REF= _control;
END_GET
END_PROPERTY

PROPERTY PowerOnPulseTask : REFERENCE TO TcoCore.TcoTask
GET
PowerOnPulseTask REF= _powerOnTask;
END_GET
END_PROPERTY

(*~
    <docu>
        <summary>
            Restores this instance to the Ready state. Can be called explicitly or from within one of the restore mechanisms.
        </summary>
    </docu>
~*)
METHOD Restore : ITcoRestorable
RestoreTasks();
_control.ActionNo := 255;
_control.GlobalSpeed := 0;
_control.ToolNo := 0;
_control.WorkobjectNo := 0;
_control.PointNo := 0;
_control.UserSpecSpeed1 := 0;
_control.UserSpecSpeed2 := 0;
_control.Coordinates.X := 0;
_control.Coordinates.Y := 0;
_control.Coordinates.Z := 0;
_control.Coordinates.Rx := 0;
_control.Coordinates.Ry := 0;
_control.Coordinates.Rz := 0;
_control.Start := FALSE;
_control.Stop := FALSE;
_control.Pause := FALSE;
_control.RunAction := FALSE;
_control.MotorOn := FALSE;
END_METHOD

METHOD INTERNAL RestoreTasks
//_resetTask.Restore();
_startAtMainTask.Restore();
_startMovementsTask.Restore();
_startProgramTask.Restore();
_startMotorsTask.Restore();
_startMotorsProgramAndMovementsTask.Restore();
_stopMovementsTask.Restore();
_startMotorsAndProgramTask.Restore();
_stopMovementsAndProgramTask.Restore();
_stopProgramTask.Restore();
_powerOnTask.Restore();
END_METHOD

(*~
    <docu>
        <summary>
            Custom service (manual, maintenance) logic.
            This method must be implemented in derived class.
        </summary>
    </docu>
~*)
METHOD PROTECTED ServiceMode
END_METHOD

PROPERTY PUBLIC SpeedSliderFraction : REFERENCE TO real
GET
SpeedSliderFraction REF= _control.Outputs.Speed.SpeedSliderFraction;
END_GET
END_PROPERTY

PROPERTY PUBLIC SSM_SpeedSliderFractionMask : REFERENCE TO BOOL
GET
SSM_SpeedSliderFractionMask REF= _control.Outputs.Speed.SSM_SpeedSliderFractionMask;
END_GET
END_PROPERTY

METHOD PUBLIC StartAtMain : TcoCore.ITcoTaskStatus
VAR_INPUT
END_VAR
StartAtMain := _startAtMainTask.Invoke();
END_METHOD

PROPERTY StartAtMainTask : TcoCore.ITcoTaskStatus
GET
StartAtMainTask := _startAtMainTask;
END_GET
END_PROPERTY

METHOD PUBLIC StartMotors : TcoCore.ITcoTaskStatus
StartMotors := _startMotorsTask.Invoke();
END_METHOD

METHOD StartMotorsAndProgram : TcoCore.ITcoTaskStatus
VAR_INPUT
END_VAR
StartMotorsAndProgram := THIS^._startMotorsAndProgramTask.Invoke();
END_METHOD

PROPERTY StartMotorsAndProgramTask : TcoCore.ITcoTaskStatus
GET
StartMotorsAndProgramTask := _startMotorsAndProgramTask;
END_GET
END_PROPERTY

METHOD PUBLIC StartMotorsProgramAndMovements : TcoCore.ITcoTaskStatus
VAR_INPUT
    inData : TcoRoboticsMovementsParams;
END_VAR
StartMotorsProgramAndMovements := _startMotorsProgramAndMovementsTask.InvokeWithParams(inData);
END_METHOD

PROPERTY StartMotorsProgramAndMovementsTask : TcoCore.ITcoTaskStatus
GET
StartMotorsProgramAndMovementsTask := _startMotorsProgramAndMovementsTask;
END_GET
END_PROPERTY

PROPERTY StartMotorsTask : TcoCore.ITcoTaskStatus
GET
StartMotorsTask := _startMotorsTask;
END_GET
END_PROPERTY

METHOD PUBLIC StartMovements : TcoCore.ITcoTaskStatus
VAR_INPUT
    inData : TcoRoboticsMovementsParams;
END_VAR
StartMovements := _startMovementsTask.InvokeWithParams(inData);
END_METHOD

PROPERTY StartMovementsTask : TcoCore.ITcoTaskStatus
GET
StartMovementsTask := _startMovementsTask;
END_GET
END_PROPERTY

METHOD PUBLIC StartProgram : TcoCore.ITcoTaskStatus
StartProgram := _startProgramTask.Invoke();
END_METHOD

PROPERTY StartProgramTask : TcoCore.ITcoTaskStatus
GET
StartProgramTask := _startProgramTask;
END_GET
END_PROPERTY

(*~
    <docu>
        <summary>
            Gets the status of the IRC5.
        </summary>
    </docu>
~*)
PROPERTY Status : REFERENCE TO TcoUrRobotics_Status_v_1_x_x
GET
Status REF= _status;
END_GET
END_PROPERTY

METHOD PUBLIC StopMovements : TcoCore.ITcoTaskStatus
VAR_INPUT
    inStopType : eTcoRoboticsStopType;
END_VAR
StopMovements := _stopMovementsTask.InvokeWithParams(inStopType);
END_METHOD

METHOD PUBLIC StopMovementsAndProgram : TcoCore.ITcoTaskStatus
VAR_INPUT
    inStopType : eTcoRoboticsStopType;
END_VAR
StopMovementsAndProgram := _stopMovementsAndProgramTask.InvokeWithParams(inStopType);
END_METHOD

PROPERTY StopMovementsAndProgramTask : TcoCore.ITcoTaskStatus
GET
StopMovementsAndProgramTask := _stopMovementsAndProgramTask;
END_GET
END_PROPERTY

PROPERTY StopMovementsTask : TcoCore.ITcoTaskStatus
GET
StopMovementsTask := _stopMovementsTask;
END_GET
END_PROPERTY

METHOD PUBLIC StopProgram : TcoCore.ITcoTaskStatus
StopProgram := _stopProgramTask.Invoke();
END_METHOD

PROPERTY StopProgramTask : TcoCore.ITcoTaskStatus
GET
StopProgramTask := _stopProgramTask;
END_GET
END_PROPERTY

METHOD INTERNAL UpdateControl
VAR_INPUT
END_VAR
VAR
    index : INT;
    offset : INT;
END_VAR
//SYSTEM OUTPUTS
index := 0;
_control.Outputs.Reg1.Bits[index] := _control.Start;
index := index + 1;
_control.outputs.Reg1.Bits[index] := _control.Stop;
index := index + 1;
_control.outputs.Reg1.Bits[index] := _control.Pause;
index := index + 1;
_control.outputs.Reg1.Bits[index] := _control.MotorOn;
index := index + 1;
//_control.outputs.Reg1.Bits[index] := _control.RunAction;
//index := index + 1;
index := 8;
//Tool signals
_control.Outputs.Reg1.Bits[index] := _control.Tool_1_Retract;
index := index + 1;
_control.outputs.Reg1.Bits[index] := _control.Tool_1_Extend;
index := index + 1;
_control.outputs.Reg1.Bits[index] := _control.Tool_2_Retract;
index := index + 1;
_control.outputs.Reg1.Bits[index] := _control.Tool_2_Extend;
index := index + 1;
_control.outputs.Reg1.Bits[index] := _control.Tool_3_Retract;
index := index + 1;
_control.outputs.Reg1.Bits[index] := _control.Tool_3_Extend;
index := index + 1;
_control.outputs.Reg1.Bits[index] := _control.Tool_4_Retract;
index := index + 1;
_control.outputs.Reg1.Bits[index] := _control.Tool_4_Extend;
index := index + 1;
//zone
index := 0;
_control.Outputs.Reg1.Ints[index] := _control.Zone;
//position
index := index + 1;
_control.Outputs.Reg1.Ints[index] := _control.InPosition;
//
//Movement parameters
index := index + 1;
_control.Outputs.Reg1.Ints[index] := _control.ActionNo;
index := index + 1;
_control.Outputs.Reg1.Ints[index] := _control.GlobalSpeed;
index := index + 1;
_control.Outputs.Reg1.Ints[index] := _control.ToolNo;
index := index + 1;
_control.Outputs.Reg1.Ints[index] := _control.WorkobjectNo;
index := index + 1;
_control.Outputs.Reg1.Ints[index] := _control.PointNo;
//master mode  such as manual/auto ....
index := index + 1;
_control.Outputs.Reg1.Ints[index] := _control.MasterMode;
index := 0;
_control.Outputs.Reg1.Floats[index] := _control.UserSpecSpeed1;
index := index + 1;
_control.Outputs.Reg1.Floats[index] := _control.UserSpecSpeed2;
index := index + 1;
////Coordinates
_control.Outputs.Reg1.Floats[index] := _control.Coordinates.X;
index := index + 1;
_control.Outputs.Reg1.Floats[index] := _control.Coordinates.Y;
index := index + 1;
_control.Outputs.Reg1.Floats[index] := _control.Coordinates.Z;
index := index + 1;
_control.Outputs.Reg1.Floats[index] := (_control.Coordinates.Rx);
index := index + 1;
_control.Outputs.Reg1.Floats[index] := (_control.Coordinates.Ry);
index := index + 1;
_control.Outputs.Reg1.Floats[index] := (_control.Coordinates.Rz);
//st_URO_CB3_O2TSpeedData => 8_O2T Robot IO
index := 0;
inoData.Out.RobotIO.bArray[index].0 := _control.Outputs.Speed.SSM_SpeedSliderFractionMask;
index := index + 4; //Reserve

TcoUtilities.TcoRealToBytes(TcoUtilities.eTcoDataFormat.BigEndian,
    _control.Outputs.Speed.SpeedSliderFraction / 100.0,
    inoData.Out.RobotIO.bArray[index],
    inoData.Out.RobotIO.bArray[index + 1],
    inoData.Out.RobotIO.bArray[index + 2],
    inoData.Out.RobotIO.bArray[index + 3]);

index := index + 4;
//st_URO_CB3_O2TIoData => 8_O2T Robot IO
inoData.Out.RobotIO.bArray[index] := _control.Outputs.IO.StandardDigitalOutputMask;
index := index + 1;
inoData.Out.RobotIO.bArray[index] := _control.Outputs.IO.ConfigurableDigitalOutputMask;
index := index + 1;
inoData.Out.RobotIO.bArray[index] := _control.Outputs.IO.StandardDigitalOutputs;
index := index + 1;
inoData.Out.RobotIO.bArray[index] := _control.Outputs.IO.ConfigurableDdigitalOutputs;
index := index + 1;
inoData.Out.RobotIO.bArray[index] := _control.Outputs.IO.AOM_AnalogOutputMask;
index := index + 1;
inoData.Out.RobotIO.bArray[index] := _control.Outputs.IO.AOT_AnalogOutputTypes;
index := index + 1;
inoData.Out.RobotIO.bArray[index] := _control.Outputs.IO.TDOM_ToolDigitalOutputMask;
index := index + 1;
inoData.Out.RobotIO.bArray[index] := _control.Outputs.IO.TDO_ToolDigitalOutput;
index := index + 1;

TcoUtilities.TcoRealToBytes(TcoUtilities.eTcoDataFormat.BigEndian,
    _control.Outputs.IO.StandardAnalogOutput[0],
    inoData.Out.RobotIO.bArray[index],
    inoData.Out.RobotIO.bArray[index + 1],
    inoData.Out.RobotIO.bArray[index + 2],
    inoData.Out.RobotIO.bArray[index + 3]);

index := index + 4;

TcoUtilities.TcoRealToBytes(TcoUtilities.eTcoDataFormat.BigEndian,
    _control.Outputs.IO.StandardAnalogOutput[1],
    inoData.Out.RobotIO.bArray[index],
    inoData.Out.RobotIO.bArray[index + 1],
    inoData.Out.RobotIO.bArray[index + 2],
    inoData.Out.RobotIO.bArray[index + 3]);

index := index + 4;
//st_URO_CB3_O2TRegData => 9_O2T General Purpose Registers 1
index := 0;

FOR offset := 0 TO 31 DO
    TcoUtilities.TcoSetBitInByte(_control.Outputs.Reg1.Bits[offset], offset MOD 8, inoData.Out.Reg1.bArray[index + (offset - (offset MOD 8)) / 8]);
END_FOR

index := index + 4;

FOR offset := 0 TO 11 DO
    TcoUtilities.TcoDintToBytes(TcoUtilities.eTcoDataFormat.BigEndian,
        _control.Outputs.Reg1.Ints[offset],
        inodata.Out.Reg1.bArray[index],
        inodata.Out.Reg1.bArray[index + 1],
        inodata.Out.Reg1.bArray[index + 2],
        inodata.Out.Reg1.bArray[index + 3]);

    index := index + 4;
END_FOR

FOR offset := 0 TO 11 DO
    TcoUtilities.TcoRealToBytes(TcoUtilities.eTcoDataFormat.BigEndian,
        _control.Outputs.Reg1.Floats[offset],
        inodata.Out.Reg1.bArray[index],
        inodata.Out.Reg1.bArray[index + 1],
        inodata.Out.Reg1.bArray[index + 2],
        inodata.Out.Reg1.bArray[index + 3]);

    index := index + 4;
END_FOR
//st_URO_CB3_O2TRegData => 10_O2T General Purpose Registers 2
index := 0;

FOR offset := 0 TO 31 DO
    TcoUtilities.TcoSetBitInByte(_control.Outputs.Reg2.Bits[offset], offset MOD 8, inoData.Out.Reg2.bArray[index + (offset - (offset MOD 8)) / 8]);
END_FOR

index := index + 4;

FOR offset := 0 TO 11 DO
    TcoUtilities.TcoDintToBytes(TcoUtilities.eTcoDataFormat.BigEndian,
        _control.Outputs.Reg2.Ints[offset],
        inodata.Out.Reg2.bArray[index],
        inodata.Out.Reg2.bArray[index + 1],
        inodata.Out.Reg2.bArray[index + 2],
        inodata.Out.Reg2.bArray[index + 3]);

    index := index + 4;
END_FOR

FOR offset := 0 TO 11 DO
    TcoUtilities.TcoRealToBytes(TcoUtilities.eTcoDataFormat.BigEndian,
        _control.Outputs.Reg2.Floats[offset],
        inodata.Out.Reg2.bArray[index],
        inodata.Out.Reg2.bArray[index + 1],
        inodata.Out.Reg2.bArray[index + 2],
        inodata.Out.Reg2.bArray[index + 3]);

    index := index + 4;
END_FOR
END_METHOD

METHOD INTERNAL UpdateStatus
VAR
    _message : STRING(125);
    tempOut : BYTE;
    index : INT;
    _bytes : DINT;
    offset : INT;
END_VAR
//Inputs Low level
//INPUTS T2O STATE ROBOT => st_URO_CB3_T2OInfoData
index := 0;
Status.State.Inputs.Robot.ControllerMajorVersion := inoData.In.State.bArray[index];
index := index + 1;
Status.State.Inputs.Robot.ControllerMinorVersion := inoData.In.State.bArray[index];
index := index + 1;
index := 4; //index + 2; //reserve
Status.State.Inputs.Robot.RobotMode := inoData.In.State.bArray[index];
index := index + 1;
Status.State.Inputs.Robot.RealtimeMachineSeconds := inoData.In.State.bArray[index];
index := index + 1;

Status.State.Inputs.Robot.RealtimeMachineMilliseconds :=
    TcoUtilities.TcoBytesToUint(TcoUtilities.eTcoDataFormat.BigEndian, inoData.In.State.bArray[index], inoData.In.State.bArray[index + 1]);
//index := index + 2;
index := 8;
Status.State.Inputs.Robot.RealtimeMachineMinutes := inoData.In.State.bArray[index];
index := index + 1;
Status.State.Inputs.Robot.RealtimeMachineHours := inoData.In.State.bArray[index];
index := index + 1;

Status.State.Inputs.Robot.RealtimeMachineDays :=
    TcoUtilities.TcoBytesToUint(TcoUtilities.eTcoDataFormat.BigEndian, inoData.In.State.bArray[index], inoData.In.State.bArray[index + 1]);
//index := index + 2;
index := 12;

Status.State.Inputs.Robot.RobotCurrent := TcoUtilities.TcoBytesToReal(TcoUtilities.eTcoDataFormat.BigEndian,
    inoData.In.State.bArray[index],
    inoData.In.State.bArray[index + 1],
    inoData.In.State.bArray[index + 2],
    inoData.In.State.bArray[index + 3]);
//index := index + 4;
index := 16;
//INPUTS T2O STATE ROBOT => st_URO_CB3_T2OStateData
Status.State.Inputs.Robot.PW_IsPowerOn := inoData.In.State.bArray[index].0;
Status.State.Inputs.Robot.PR_IsProgramRunning := inoData.In.State.bArray[index].1;
Status.State.Inputs.Robot.TB_IsTeachButtonPressed := inoData.In.State.bArray[index].2;
Status.State.Inputs.Robot.PB_IsPowerButtonPressed := inoData.In.State.bArray[index].3;
index := 20;

Status.State.Inputs.Robot.SpeedSliderFraction := 100 *
    TcoUtilities.TcoBytesToReal(TcoUtilities.eTcoDataFormat.BigEndian,
        inoData.In.State.bArray[index],
        inoData.In.State.bArray[index + 1],
        inoData.In.State.bArray[index + 2],
        inoData.In.State.bArray[index + 3]);
//index := index + 4;
index := 24;
Status.State.Inputs.Safety.SafetyMode := inoData.In.State.bArray[index];
//index := index + 1;
index := 28;
Status.State.Inputs.Safety.NO_IsNormalMode := inoData.In.State.bArray[index].0;
Status.State.Inputs.Safety.RD_IsReducedMode := inoData.In.State.bArray[index].1;
Status.State.Inputs.Safety.PS_IsProtectiveStopped := inoData.In.State.bArray[index].2;
Status.State.Inputs.Safety.RC_IsRecoveryMode := inoData.In.State.bArray[index].3;
Status.State.Inputs.Safety.SS_IsSafeguardStopped := inoData.In.State.bArray[index].4;
Status.State.Inputs.Safety.SES_IsSystemEmergencyStopped := inoData.In.State.bArray[index].5;
Status.State.Inputs.Safety.RES_IsRobotEmergencyStopped := inoData.In.State.bArray[index].6;
Status.State.Inputs.Safety.ES_IsEmergencyStopped := inoData.In.State.bArray[index].7;
index := index + 1;
Status.State.Inputs.Safety.VL_IsViolation := inoData.In.State.bArray[index].0;
Status.State.Inputs.Safety.FT_IsFault := inoData.In.State.bArray[index].1;
Status.State.Inputs.Safety.ST_IsStoppedDueSafety := inoData.In.State.bArray[index].2;
//INPUTS T20 IO => st_URO_CB3_T2OIoStateData
index := 0;
Status.State.Inputs.IO.StandardDigitalInputs := inoData.In.IO.bArray[index];
index := index + 1;
Status.State.Inputs.IO.ConfigurableDigitalInputs := inoData.In.IO.bArray[index];
index := index + 1;
Status.State.Inputs.IO.StandardDigitalOutputs := inoData.In.IO.bArray[index];
index := index + 1;
Status.State.Inputs.IO.ConfigurableDigitalOutputs := inoData.In.IO.bArray[index];
Index := 4;
Status.State.Inputs.IO.AnalogIoTypes := inoData.In.IO.bArray[index];
index := index + 1;
index := 8; //reserve

Status.State.Inputs.IO.StandardAnalogInput[0] := TcoUtilities.TcoBytesToReal(TcoUtilities.eTcoDataFormat.BigEndian,
    inoData.In.IO.bArray[index],
    inoData.In.IO.bArray[index + 1],
    inoData.In.IO.bArray[index + 2],
    inoData.In.IO.bArray[index + 3]);

index := index + 4;

Status.State.Inputs.IO.StandardAnalogInput[1] := TcoUtilities.TcoBytesToReal(TcoUtilities.eTcoDataFormat.BigEndian,
    inoData.In.IO.bArray[index],
    inoData.In.IO.bArray[index + 1],
    inoData.In.IO.bArray[index + 2],
    inoData.In.IO.bArray[index + 3]);

index := index + 4;

Status.State.Inputs.IO.StandardAnalogOutput[0] := TcoUtilities.TcoBytesToReal(TcoUtilities.eTcoDataFormat.BigEndian,
    inoData.In.IO.bArray[index],
    inoData.In.IO.bArray[index + 1],
    inoData.In.IO.bArray[index + 2],
    inoData.In.IO.bArray[index + 3]);

index := index + 4;

Status.State.Inputs.IO.StandardAnalogOutput[1] := TcoUtilities.TcoBytesToReal(TcoUtilities.eTcoDataFormat.BigEndian,
    inoData.In.IO.bArray[index],
    inoData.In.IO.bArray[index + 1],
    inoData.In.IO.bArray[index + 2],
    inoData.In.IO.bArray[index + 3]);

index := index + 4;

Status.State.Inputs.IO.Current := TcoUtilities.TcoBytesToReal(TcoUtilities.eTcoDataFormat.BigEndian,
    inoData.In.IO.bArray[index],
    inoData.In.IO.bArray[index + 1],
    inoData.In.IO.bArray[index + 2],
    inoData.In.IO.bArray[index + 3]);

index := index + 4;

FOR offset := 0 TO 7 DO
    Status.State.Inputs.IO.Euromap67InputBits[offset] := TcoUtilities.TcoGetBitFromByte(inoData.In.IO.bArray[index], offset);
    Status.State.Inputs.IO.Euromap67InputBits[offset + 8] := TcoUtilities.TcoGetBitFromByte(inoData.In.IO.bArray[index + 1], offset);
    Status.State.Inputs.IO.Euromap67InputBits[offset + 16] := TcoUtilities.TcoGetBitFromByte(inoData.In.IO.bArray[index + 2], offset);
    Status.State.Inputs.IO.Euromap67InputBits[offset + 24] := TcoUtilities.TcoGetBitFromByte(inoData.In.IO.bArray[index + 3], offset);
END_FOR

index := index + 4;

FOR offset := 0 TO 7 DO
    Status.State.Inputs.IO.Euromap67OutputBits[offset] := TcoUtilities.TcoGetBitFromByte(inoData.In.IO.bArray[index], offset);
    Status.State.Inputs.IO.Euromap67OutputBits[offset + 8] := TcoUtilities.TcoGetBitFromByte(inoData.In.IO.bArray[index + 1], offset);
    Status.State.Inputs.IO.Euromap67OutputBits[offset + 16] := TcoUtilities.TcoGetBitFromByte(inoData.In.IO.bArray[index + 2], offset);
    Status.State.Inputs.IO.Euromap67OutputBits[offset + 24] := TcoUtilities.TcoGetBitFromByte(inoData.In.IO.bArray[index + 3], offset);
END_FOR

index := index + 4;

Status.State.Inputs.IO.Euromap6724Voltage := TcoUtilities.TcoBytesToReal(TcoUtilities.eTcoDataFormat.BigEndian,
    inoData.In.IO.bArray[index],
    inoData.In.IO.bArray[index + 1],
    inoData.In.IO.bArray[index + 2],
    inoData.In.IO.bArray[index + 3]);

index := index + 4;

Status.State.Inputs.IO.Euromap6724VCurrent := TcoUtilities.TcoBytesToReal(TcoUtilities.eTcoDataFormat.BigEndian,
    inoData.In.IO.bArray[index],
    inoData.In.IO.bArray[index + 1],
    inoData.In.IO.bArray[index + 2],
    inoData.In.IO.bArray[index + 3]);

index := index + 4;
//INPUTS T20 IO => st_URO_CB3_T2OToolStateData
Status.State.Inputs.Tool.ToolMode := inoData.In.IO.bArray[index];
index := index + 1;
Status.State.Inputs.Tool.TDI_ToolDigitalInputs := inoData.In.IO.bArray[index];
index := index + 1;
Status.State.Inputs.Tool.TDO_ToolDigitalOutputs := inoData.In.IO.bArray[index];
index := index + 1;
Status.State.Inputs.Tool.TAIT_ToolAnalogInputTypes := inoData.In.IO.bArray[index];
index := index + 1;

Status.State.Inputs.Tool.ToolAnalogInput[0] := TcoUtilities.TcoBytesToReal(TcoUtilities.eTcoDataFormat.BigEndian,
    inoData.In.IO.bArray[index],
    inoData.In.IO.bArray[index + 1],
    inoData.In.IO.bArray[index + 2],
    inoData.In.IO.bArray[index + 3]);

index := index + 4;

Status.State.Inputs.Tool.ToolAnalogInput[1] := TcoUtilities.TcoBytesToReal(TcoUtilities.eTcoDataFormat.BigEndian,
    inoData.In.IO.bArray[index],
    inoData.In.IO.bArray[index + 1],
    inoData.In.IO.bArray[index + 2],
    inoData.In.IO.bArray[index + 3]);

index := index + 4;

Status.State.Inputs.Tool.ToolOutputVoltage := TcoUtilities.TcoBytesToReal(TcoUtilities.eTcoDataFormat.BigEndian,
    inoData.In.IO.bArray[index],
    inoData.In.IO.bArray[index + 1],
    inoData.In.IO.bArray[index + 2],
    inoData.In.IO.bArray[index + 3]);

index := index + 4;

Status.State.Inputs.Tool.ToolCurrent := TcoUtilities.TcoBytesToReal(TcoUtilities.eTcoDataFormat.BigEndian,
    inoData.In.IO.bArray[index],
    inoData.In.IO.bArray[index + 1],
    inoData.In.IO.bArray[index + 2],
    inoData.In.IO.bArray[index + 3]);

index := index + 4;
//INPUTS T20 JOINT => st_URO_CB3_T2OJointsData
index := 0;

Status.State.Inputs.Joints.JointPosition[0] := RAD_TO_DEG(TcoUtilities.TcoBytesToReal(TcoUtilities.eTcoDataFormat.BigEndian,
        inoData.In.Joints.bArray[index],
        inoData.In.Joints.bArray[index + 1],
        inoData.In.Joints.bArray[index + 2],
        inoData.In.Joints.bArray[index + 3]));

index := index + 4;

Status.State.Inputs.Joints.JointPosition[1] := RAD_TO_DEG(TcoUtilities.TcoBytesToReal(TcoUtilities.eTcoDataFormat.BigEndian,
        inoData.In.Joints.bArray[index],
        inoData.In.Joints.bArray[index + 1],
        inoData.In.Joints.bArray[index + 2],
        inoData.In.Joints.bArray[index + 3]));

index := index + 4;

Status.State.Inputs.Joints.JointPosition[2] := RAD_TO_DEG(TcoUtilities.TcoBytesToReal(TcoUtilities.eTcoDataFormat.BigEndian,
        inoData.In.Joints.bArray[index],
        inoData.In.Joints.bArray[index + 1],
        inoData.In.Joints.bArray[index + 2],
        inoData.In.Joints.bArray[index + 3]));

index := index + 4;

Status.State.Inputs.Joints.JointPosition[3] := RAD_TO_DEG(TcoUtilities.TcoBytesToReal(TcoUtilities.eTcoDataFormat.BigEndian,
        inoData.In.Joints.bArray[index],
        inoData.In.Joints.bArray[index + 1],
        inoData.In.Joints.bArray[index + 2],
        inoData.In.Joints.bArray[index + 3]));

index := index + 4;

Status.State.Inputs.Joints.JointPosition[4] := RAD_TO_DEG(TcoUtilities.TcoBytesToReal(TcoUtilities.eTcoDataFormat.BigEndian,
        inoData.In.Joints.bArray[index],
        inoData.In.Joints.bArray[index + 1],
        inoData.In.Joints.bArray[index + 2],
        inoData.In.Joints.bArray[index + 3]));

index := index + 4;

Status.State.Inputs.Joints.JointPosition[5] := RAD_TO_DEG(TcoUtilities.TcoBytesToReal(TcoUtilities.eTcoDataFormat.BigEndian,
        inoData.In.Joints.bArray[index],
        inoData.In.Joints.bArray[index + 1],
        inoData.In.Joints.bArray[index + 2],
        inoData.In.Joints.bArray[index + 3]));

index := index + 4;

Status.State.Inputs.Joints.JointVelocity[0] := TcoUtilities.TcoBytesToReal(TcoUtilities.eTcoDataFormat.BigEndian,
    inoData.In.Joints.bArray[index],
    inoData.In.Joints.bArray[index + 1],
    inoData.In.Joints.bArray[index + 2],
    inoData.In.Joints.bArray[index + 3]);

index := index + 4;

Status.State.Inputs.Joints.JointVelocity[1] := TcoUtilities.TcoBytesToReal(TcoUtilities.eTcoDataFormat.BigEndian,
    inoData.In.Joints.bArray[index],
    inoData.In.Joints.bArray[index + 1],
    inoData.In.Joints.bArray[index + 2],
    inoData.In.Joints.bArray[index + 3]);

index := index + 4;

Status.State.Inputs.Joints.JointVelocity[2] := TcoUtilities.TcoBytesToReal(TcoUtilities.eTcoDataFormat.BigEndian,
    inoData.In.Joints.bArray[index],
    inoData.In.Joints.bArray[index + 1],
    inoData.In.Joints.bArray[index + 2],
    inoData.In.Joints.bArray[index + 3]);

index := index + 4;

Status.State.Inputs.Joints.JointVelocity[3] := TcoUtilities.TcoBytesToReal(TcoUtilities.eTcoDataFormat.BigEndian,
    inoData.In.Joints.bArray[index],
    inoData.In.Joints.bArray[index + 1],
    inoData.In.Joints.bArray[index + 2],
    inoData.In.Joints.bArray[index + 3]);

index := index + 4;

Status.State.Inputs.Joints.JointVelocity[4] := TcoUtilities.TcoBytesToReal(TcoUtilities.eTcoDataFormat.BigEndian,
    inoData.In.Joints.bArray[index],
    inoData.In.Joints.bArray[index + 1],
    inoData.In.Joints.bArray[index + 2],
    inoData.In.Joints.bArray[index + 3]);

index := index + 4;

Status.State.Inputs.Joints.JointVelocity[5] := TcoUtilities.TcoBytesToReal(TcoUtilities.eTcoDataFormat.BigEndian,
    inoData.In.Joints.bArray[index],
    inoData.In.Joints.bArray[index + 1],
    inoData.In.Joints.bArray[index + 2],
    inoData.In.Joints.bArray[index + 3]);

index := index + 4;

Status.State.Inputs.Joints.JointCurrent[0] := TcoUtilities.TcoBytesToReal(TcoUtilities.eTcoDataFormat.BigEndian,
    inoData.In.Joints.bArray[index],
    inoData.In.Joints.bArray[index + 1],
    inoData.In.Joints.bArray[index + 2],
    inoData.In.Joints.bArray[index + 3]);

index := index + 4;

Status.State.Inputs.Joints.JointCurrent[1] := TcoUtilities.TcoBytesToReal(TcoUtilities.eTcoDataFormat.BigEndian,
    inoData.In.Joints.bArray[index],
    inoData.In.Joints.bArray[index + 1],
    inoData.In.Joints.bArray[index + 2],
    inoData.In.Joints.bArray[index + 3]);

index := index + 4;

Status.State.Inputs.Joints.JointCurrent[2] := TcoUtilities.TcoBytesToReal(TcoUtilities.eTcoDataFormat.BigEndian,
    inoData.In.Joints.bArray[index],
    inoData.In.Joints.bArray[index + 1],
    inoData.In.Joints.bArray[index + 2],
    inoData.In.Joints.bArray[index + 3]);

index := index + 4;

Status.State.Inputs.Joints.JointCurrent[3] := TcoUtilities.TcoBytesToReal(TcoUtilities.eTcoDataFormat.BigEndian,
    inoData.In.Joints.bArray[index],
    inoData.In.Joints.bArray[index + 1],
    inoData.In.Joints.bArray[index + 2],
    inoData.In.Joints.bArray[index + 3]);

index := index + 4;

Status.State.Inputs.Joints.JointCurrent[4] := TcoUtilities.TcoBytesToReal(TcoUtilities.eTcoDataFormat.BigEndian,
    inoData.In.Joints.bArray[index],
    inoData.In.Joints.bArray[index + 1],
    inoData.In.Joints.bArray[index + 2],
    inoData.In.Joints.bArray[index + 3]);

index := index + 4;

Status.State.Inputs.Joints.JointCurrent[5] := TcoUtilities.TcoBytesToReal(TcoUtilities.eTcoDataFormat.BigEndian,
    inoData.In.Joints.bArray[index],
    inoData.In.Joints.bArray[index + 1],
    inoData.In.Joints.bArray[index + 2],
    inoData.In.Joints.bArray[index + 3]);

index := index + 4;

Status.State.Inputs.Joints.JointTemperature[0] := TcoUtilities.TcoBytesToReal(TcoUtilities.eTcoDataFormat.BigEndian,
    inoData.In.Joints.bArray[index],
    inoData.In.Joints.bArray[index + 1],
    inoData.In.Joints.bArray[index + 2],
    inoData.In.Joints.bArray[index + 3]);

index := index + 4;

Status.State.Inputs.Joints.JointTemperature[1] := TcoUtilities.TcoBytesToReal(TcoUtilities.eTcoDataFormat.BigEndian,
    inoData.In.Joints.bArray[index],
    inoData.In.Joints.bArray[index + 1],
    inoData.In.Joints.bArray[index + 2],
    inoData.In.Joints.bArray[index + 3]);

index := index + 4;

Status.State.Inputs.Joints.JointTemperature[2] := TcoUtilities.TcoBytesToReal(TcoUtilities.eTcoDataFormat.BigEndian,
    inoData.In.Joints.bArray[index],
    inoData.In.Joints.bArray[index + 1],
    inoData.In.Joints.bArray[index + 2],
    inoData.In.Joints.bArray[index + 3]);

index := index + 4;

Status.State.Inputs.Joints.JointTemperature[3] := TcoUtilities.TcoBytesToReal(TcoUtilities.eTcoDataFormat.BigEndian,
    inoData.In.Joints.bArray[index],
    inoData.In.Joints.bArray[index + 1],
    inoData.In.Joints.bArray[index + 2],
    inoData.In.Joints.bArray[index + 3]);

index := index + 4;

Status.State.Inputs.Joints.JointTemperature[4] := TcoUtilities.TcoBytesToReal(TcoUtilities.eTcoDataFormat.BigEndian,
    inoData.In.Joints.bArray[index],
    inoData.In.Joints.bArray[index + 1],
    inoData.In.Joints.bArray[index + 2],
    inoData.In.Joints.bArray[index + 3]);

index := index + 4;

Status.State.Inputs.Joints.JointTemperature[5] := TcoUtilities.TcoBytesToReal(TcoUtilities.eTcoDataFormat.BigEndian,
    inoData.In.Joints.bArray[index],
    inoData.In.Joints.bArray[index + 1],
    inoData.In.Joints.bArray[index + 2],
    inoData.In.Joints.bArray[index + 3]);

index := index + 4;
Status.State.Inputs.Joints.JointMode[0] := inoData.In.Joints.bArray[index];
index := index + 1;
Status.State.Inputs.Joints.JointMode[1] := inoData.In.Joints.bArray[index];
index := index + 1;
Status.State.Inputs.Joints.JointMode[2] := inoData.In.Joints.bArray[index];
index := index + 1;
Status.State.Inputs.Joints.JointMode[3] := inoData.In.Joints.bArray[index];
index := index + 1;
Status.State.Inputs.Joints.JointMode[4] := inoData.In.Joints.bArray[index];
index := index + 1;
Status.State.Inputs.Joints.JointMode[5] := inoData.In.Joints.bArray[index];
index := index + 1;
//INPUTS T20 TCP => st_URO_CB3_T2OTcpData
index := 0;

Status.State.Inputs.TCP.Postition.X := 1000.0 *
    TcoUtilities.TcoBytesToReal(TcoUtilities.eTcoDataFormat.BigEndian,
        inoData.In.TCP.bArray[index],
        inoData.In.TCP.bArray[index + 1],
        inoData.In.TCP.bArray[index + 2],
        inoData.In.TCP.bArray[index + 3]);

index := index + 4;

Status.State.Inputs.TCP.Postition.Y := 1000.0 *
    TcoUtilities.TcoBytesToReal(TcoUtilities.eTcoDataFormat.BigEndian,
        inoData.In.TCP.bArray[index],
        inoData.In.TCP.bArray[index + 1],
        inoData.In.TCP.bArray[index + 2],
        inoData.In.TCP.bArray[index + 3]);

index := index + 4;

Status.State.Inputs.TCP.Postition.Z := 1000.0 *
    TcoUtilities.TcoBytesToReal(TcoUtilities.eTcoDataFormat.BigEndian,
        inoData.In.TCP.bArray[index],
        inoData.In.TCP.bArray[index + 1],
        inoData.In.TCP.bArray[index + 2],
        inoData.In.TCP.bArray[index + 3]);

index := index + 4;

Status.State.Inputs.TCP.Postition.Rx := TcoUtilities.TcoBytesToReal(TcoUtilities.eTcoDataFormat.BigEndian,
    inoData.In.TCP.bArray[index],
    inoData.In.TCP.bArray[index + 1],
    inoData.In.TCP.bArray[index + 2],
    inoData.In.TCP.bArray[index + 3]);

index := index + 4;

Status.State.Inputs.TCP.Postition.Ry := TcoUtilities.TcoBytesToReal(TcoUtilities.eTcoDataFormat.BigEndian,
    inoData.In.TCP.bArray[index],
    inoData.In.TCP.bArray[index + 1],
    inoData.In.TCP.bArray[index + 2],
    inoData.In.TCP.bArray[index + 3]);

index := index + 4;

Status.State.Inputs.TCP.Postition.Rz := TcoUtilities.TcoBytesToReal(TcoUtilities.eTcoDataFormat.BigEndian,
    inoData.In.TCP.bArray[index],
    inoData.In.TCP.bArray[index + 1],
    inoData.In.TCP.bArray[index + 2],
    inoData.In.TCP.bArray[index + 3]);

index := index + 4;

Status.State.Inputs.TCP.Velocity.X := 1000.0 *
    TcoUtilities.TcoBytesToReal(TcoUtilities.eTcoDataFormat.BigEndian,
        inoData.In.TCP.bArray[index],
        inoData.In.TCP.bArray[index + 1],
        inoData.In.TCP.bArray[index + 2],
        inoData.In.TCP.bArray[index + 3]);

index := index + 4;

Status.State.Inputs.TCP.Velocity.Y := 1000.0 *
    TcoUtilities.TcoBytesToReal(TcoUtilities.eTcoDataFormat.BigEndian,
        inoData.In.TCP.bArray[index],
        inoData.In.TCP.bArray[index + 1],
        inoData.In.TCP.bArray[index + 2],
        inoData.In.TCP.bArray[index + 3]);

index := index + 4;

Status.State.Inputs.TCP.Velocity.Z := 1000.0 *
    TcoUtilities.TcoBytesToReal(TcoUtilities.eTcoDataFormat.BigEndian,
        inoData.In.TCP.bArray[index],
        inoData.In.TCP.bArray[index + 1],
        inoData.In.TCP.bArray[index + 2],
        inoData.In.TCP.bArray[index + 3]);

index := index + 4;

Status.State.Inputs.TCP.Velocity.Rx := TcoUtilities.TcoBytesToReal(TcoUtilities.eTcoDataFormat.BigEndian,
    inoData.In.TCP.bArray[index],
    inoData.In.TCP.bArray[index + 1],
    inoData.In.TCP.bArray[index + 2],
    inoData.In.TCP.bArray[index + 3]);

index := index + 4;

Status.State.Inputs.TCP.Velocity.Ry := TcoUtilities.TcoBytesToReal(TcoUtilities.eTcoDataFormat.BigEndian,
    inoData.In.TCP.bArray[index],
    inoData.In.TCP.bArray[index + 1],
    inoData.In.TCP.bArray[index + 2],
    inoData.In.TCP.bArray[index + 3]);

index := index + 4;

Status.State.Inputs.TCP.Velocity.Rz := TcoUtilities.TcoBytesToReal(TcoUtilities.eTcoDataFormat.BigEndian,
    inoData.In.TCP.bArray[index],
    inoData.In.TCP.bArray[index + 1],
    inoData.In.TCP.bArray[index + 2],
    inoData.In.TCP.bArray[index + 3]);

index := index + 4;

Status.State.Inputs.TCP.Force.X := TcoUtilities.TcoBytesToReal(TcoUtilities.eTcoDataFormat.BigEndian,
    inoData.In.TCP.bArray[index],
    inoData.In.TCP.bArray[index + 1],
    inoData.In.TCP.bArray[index + 2],
    inoData.In.TCP.bArray[index + 3]);

index := index + 4;

Status.State.Inputs.TCP.Force.Y := TcoUtilities.TcoBytesToReal(TcoUtilities.eTcoDataFormat.BigEndian,
    inoData.In.TCP.bArray[index],
    inoData.In.TCP.bArray[index + 1],
    inoData.In.TCP.bArray[index + 2],
    inoData.In.TCP.bArray[index + 3]);

index := index + 4;

Status.State.Inputs.TCP.Force.Z := TcoUtilities.TcoBytesToReal(TcoUtilities.eTcoDataFormat.BigEndian,
    inoData.In.TCP.bArray[index],
    inoData.In.TCP.bArray[index + 1],
    inoData.In.TCP.bArray[index + 2],
    inoData.In.TCP.bArray[index + 3]);

index := index + 4;

Status.State.Inputs.TCP.Torque.X := TcoUtilities.TcoBytesToReal(TcoUtilities.eTcoDataFormat.BigEndian,
    inoData.In.TCP.bArray[index],
    inoData.In.TCP.bArray[index + 1],
    inoData.In.TCP.bArray[index + 2],
    inoData.In.TCP.bArray[index + 3]);

index := index + 4;

Status.State.Inputs.TCP.Torque.Y := TcoUtilities.TcoBytesToReal(TcoUtilities.eTcoDataFormat.BigEndian,
    inoData.In.TCP.bArray[index],
    inoData.In.TCP.bArray[index + 1],
    inoData.In.TCP.bArray[index + 2],
    inoData.In.TCP.bArray[index + 3]);

index := index + 4;

Status.State.Inputs.TCP.Torque.Z := TcoUtilities.TcoBytesToReal(TcoUtilities.eTcoDataFormat.BigEndian,
    inoData.In.TCP.bArray[index],
    inoData.In.TCP.bArray[index + 1],
    inoData.In.TCP.bArray[index + 2],
    inoData.In.TCP.bArray[index + 3]);

index := index + 4;

Status.State.Inputs.TCP.TCP_ForceScalar := TcoUtilities.TcoBytesToReal(TcoUtilities.eTcoDataFormat.BigEndian,
    inoData.In.TCP.bArray[index],
    inoData.In.TCP.bArray[index + 1],
    inoData.In.TCP.bArray[index + 2],
    inoData.In.TCP.bArray[index + 3]);

index := index + 4;
//INPUTS T20 BITS => st_URO_CB3_T2OBitRegsData
index := 0;

FOR offset := 0 TO 7 DO
    Status.State.Inputs.Bits.Register[offset] := TcoUtilities.TcoGetBitFromByte(inoData.In.BitRegs.bArray[index], offset);
    Status.State.Inputs.Bits.Register[offset + 8] := TcoUtilities.TcoGetBitFromByte(inoData.In.BitRegs.bArray[index + 1], offset);
    Status.State.Inputs.Bits.Register[offset + 16] := TcoUtilities.TcoGetBitFromByte(inoData.In.BitRegs.bArray[index + 2], offset);
    Status.State.Inputs.Bits.Register[offset + 24] := TcoUtilities.TcoGetBitFromByte(inoData.In.BitRegs.bArray[index + 3], offset);
    Status.State.Inputs.Bits.Register[offset + 32] := TcoUtilities.TcoGetBitFromByte(inoData.In.BitRegs.bArray[index + 4], offset);
    Status.State.Inputs.Bits.Register[offset + 40] := TcoUtilities.TcoGetBitFromByte(inoData.In.BitRegs.bArray[index + 5], offset);
    Status.State.Inputs.Bits.Register[offset + 48] := TcoUtilities.TcoGetBitFromByte(inoData.In.BitRegs.bArray[index + 6], offset);
    Status.State.Inputs.Bits.Register[offset + 56] := TcoUtilities.TcoGetBitFromByte(inoData.In.BitRegs.bArray[index + 7], offset);
END_FOR
//INPUTS T20 BITS => st_URO_CB3_T2OIntRegsData
index := 0;

FOR offset := 0 TO 23 DO
    Status.State.Inputs.Ints.Register[offset] := TcoUtilities.TcoBytesToDint(TcoUtilities.eTcoDataFormat.BigEndian,
        inoData.In.IntRegs.bArray[index],
        inoData.In.IntRegs.bArray[index + 1],
        inoData.In.IntRegs.bArray[index + 2],
        inoData.In.IntRegs.bArray[index + 3]);

    index := index + 4;
END_FOR
//INPUTS T20 BITS => st_URO_CB3_T2OFloatRegsData
index := 0;

FOR offset := 0 TO 23 DO
    Status.State.Inputs.Floats.Register[offset] := TcoUtilities.TcoBytesToReal(TcoUtilities.eTcoDataFormat.BigEndian,
        inoData.In.FloatRegs.bArray[index],
        inoData.In.FloatRegs.bArray[index + 1],
        inoData.In.FloatRegs.bArray[index + 2],
        inoData.In.FloatRegs.bArray[index + 3]);

    index := index + 4;
END_FOR

_status.State.RobotMode := GetRobotModeDescription(_status.State.Inputs.Robot.RobotMode);
//SYSTEM INPUTS
index := 0;
//Area/positions flags this  should be obsolete because Zones and InPosition is used as byte below
index := 0;
_status.State.InArea_1 := _status.State.Inputs.Bits.Register[index];
index := index + 1;
_status.State.InArea_2 := _status.State.Inputs.Bits.Register[index];
index := index + 1;
_status.State.InArea_3 := _status.State.Inputs.Bits.Register[index];
index := index + 1;
_status.State.InArea_4 := _status.State.Inputs.Bits.Register[index];
index := index + 1;
_status.State.InPosition_1 := _status.State.Inputs.Bits.Register[index];
index := index + 1;
_status.State.InPosition_2 := _status.State.Inputs.Bits.Register[index];
index := index + 1;
_status.State.InPosition_3 := _status.State.Inputs.Bits.Register[index];
index := index + 1;
_status.State.InPosition_4 := _status.State.Inputs.Bits.Register[index];
index := index + 1;
//
//Tool signals
_status.State.Tool_1_Retract := _status.State.Inputs.Bits.Register[index];
index := index + 1;
_status.State.Tool_1_Extend := _status.State.Inputs.Bits.Register[index];
index := index + 1;
_status.State.Tool_2_Retract := _status.State.Inputs.Bits.Register[index];
index := index + 1;
_status.State.Tool_2_Extend := _status.State.Inputs.Bits.Register[index];
index := index + 1;
_status.State.Tool_3_Retract := _status.State.Inputs.Bits.Register[index];
index := index + 1;
_status.State.Tool_3_Extend := _status.State.Inputs.Bits.Register[index];
index := index + 1;
_status.State.Tool_4_Retract := _status.State.Inputs.Bits.Register[index];
index := index + 1;
_status.State.Tool_4_Extend := _status.State.Inputs.Bits.Register[index];
index := index + 1;
index := 0;
_status.State.Zone := _status.State.Inputs.Ints.Register[index];
index := index + 1;
_status.State.InPosition := _status.State.Inputs.Ints.Register[index];
//Movement parameters
index := index + 1;
_status.State.ActionNo := _status.State.Inputs.Ints.Register[index];
index := index + 1;
_status.State.GlobalSpeed := _status.State.Inputs.Ints.Register[index];
index := index + 1;
_status.State.ToolNo := _status.State.Inputs.Ints.Register[index];
index := index + 1;
_status.State.WorkobjectNo := _status.State.Inputs.Ints.Register[index];
index := index + 1;
_status.State.PointNo := _status.State.Inputs.Ints.Register[index];
index := index + 1;
index := 0;
_status.State.UserSpecSpeed1 := _status.State.Inputs.Floats.Register[index];
index := index + 1;
_status.State.UserSpecSpeed2 := _status.State.Inputs.Floats.Register[index];
index := index + 1;
_status.State.Coordinates.X := Status.State.Inputs.Floats.Register[index];
index := index + 1;
_status.State.Coordinates.Y := Status.State.Inputs.Floats.Register[index];
index := index + 1;
_status.State.Coordinates.Z := Status.State.Inputs.Floats.Register[index];
index := index + 1;
_status.State.Coordinates.Rx := Status.State.Inputs.Floats.Register[index];
index := index + 1;
_status.State.Coordinates.Ry := Status.State.Inputs.Floats.Register[index];
index := index + 1;
_status.State.Coordinates.Rz := Status.State.Inputs.Floats.Register[index];
index := index + 1;
//toido event id
END_METHOD

END_FUNCTION_BLOCK

// ---- POUs/Prototypes/RoboticsTasks/Starts/StartAtMainTask.TcPOU
FUNCTION_BLOCK StartAtMainTask EXTENDS TcoUrRoboticsTask

IF Execute() THEN
    _blink(inOnTime := T#500MS, inOffTime := T#500MS);

    IF _progress = 0 THEN
        IF NOT __ISVALIDREF(inoControl) THEN
            _varInfo := __VARINFO(inoControl);
            Messenger.Programming(_sb.Clear().Append('<#Invalid reference: #>').Append(_varInfo.Symbol).ToString()).Pin();
        ELSIF NOT __ISVALIDREF(inoConfig) THEN
            _varInfo := __VARINFO(inoConfig);
            Messenger.Programming(_sb.Clear().Append('<#Invalid reference: #>').Append(_varInfo.Symbol).ToString()).Pin();
        ELSIF NOT __ISVALIDREF(inoStatus) THEN
            _varInfo := __VARINFO(inoStatus);
            Messenger.Programming(_sb.Clear().Append('<#Invalid reference: #>').Append(_varInfo.Symbol).ToString()).Pin();
        ELSE
            _progress := _progress + 1;
        END_IF
    END_IF

    IF _progress = 1 THEN
        THIS^.Messenger.OnCondition(_infoTimer.Q AND NOT inoStatus.State.Inputs.Safety.NO_IsNormalMode)
            .Warning(_sb.Clear().Append('<# Waiting to Normal Mode. #>').ToString());

        THIS^.Messenger.OnCondition(_infoTimer.Q AND NOT inoStatus.State.Inputs.Safety.RD_IsReducedMode)
            .Warning(_sb.Clear().Append('<# Waiting to Reduced Mode. #>').ToString());

        IF inoStatus.State.Inputs.Safety.NO_IsNormalMode OR inoStatus.State.Inputs.Safety.RD_IsReducedMode THEN
            _progress := _progress + 1;
        END_IF
    END_IF;

    IF _progress = 2 THEN
        inoControl.Start := _blink.outQ;

        THIS^.Messenger.OnCondition(_infoTimer.Q AND NOT inoStatus.State.Inputs.Robot.PR_IsProgramRunning)
            .Warning(_sb.Clear().Append('<#Waiting to program running! #>').ToString());

        IF inoStatus.State.Inputs.Robot.PR_IsProgramRunning THEN
            inoControl.Start := FALSE;
            _progress := 0;
        END_IF
    END_IF

    DoneWhen(inoStatus.State.Inputs.Robot.PR_IsProgramRunning);
    CallTimers(TRUE);
    THIS^.ThrowWhen(_errorTimer.Q);
END_IF;

IF THIS^.Error AND NOT _errorMessage.Pinned THEN
    THIS^.Restore();
END_IF

(*~
    <docu>
        <summary>
            Executes when task is aborted.
        </summary>
    </docu>
~*)
METHOD PROTECTED OnAbort
IF __ISVALIDREF(inoStatus) THEN
    THIS^.inoStatus.ActionDescription := '<#Start at Main was aborted, while not yet completed!#>';
END_IF;
END_METHOD

(*~
    <docu>
        <summary>
            Executes when task reaches the ```Done``` state .
        </summary>
    </docu>
~*)
METHOD PROTECTED OnDone
IF __ISVALIDREF(inoStatus) THEN
    THIS^.inoStatus.ActionDescription := '<#Start at Main was completed successfully.#>';
END_IF;
END_METHOD

(*~
    <docu>
        <summary>
            Executes when task reaches the ```Error``` state.
            <para>
                Do not confuse with <see cref="PlcDocu.TcoCore.TcoTask.WhileError()"/>, that is called cyclically until '''Error''' state is left.
            </para>
        </summary>
    </docu>
~*)
METHOD PROTECTED OnError
VAR
    description : STRING;
END_VAR
description := '<#Start at Main finished with error.#>';

IF __ISVALIDREF(inoStatus) THEN
    THIS^.inoStatus.ActionDescription := description;
END_IF;

THIS^._errorMessage.Error(_sb.Clear().Append(description).Append(' To restore acknowledge this alarm.').ToString()).Pin();
END_METHOD

METHOD PROTECTED OnStart
IF __ISVALIDREF(inoStatus) THEN
    THIS^.inoStatus.ActionDescription := '<#Start at Main started.#>';
END_IF;

CallTimers(FALSE);
END_METHOD

(*~
    <docu>
        <summary>
            Restores this instance to the Ready state. Can be called explicitly or from within one of the restore mechanisms.
            <para>
                See also <see cref="PlcDocu.TcoCore.TcoTask.AutoRestorable()"/>
            </para>
        </summary>
    </docu>
~*)
METHOD Restore : ITcoRestorable
SUPER^.Restore();
END_METHOD

END_FUNCTION_BLOCK

// ---- POUs/Prototypes/RoboticsTasks/TcoUrRoboticsTask.TcPOU
FUNCTION_BLOCK PUBLIC ABSTRACT TcoUrRoboticsTask EXTENDS TcoCore.TcoTask
VAR_IN_OUT
    inoConfig : TcoUrRobotics_Config_v_1_x_x;
    inoControl : TcoUrRobotics_Control_v_1_x_x;
    inoStatus : TcoUrRobotics_Status_v_1_x_x;
END_VAR
VAR
    _errorMessage : TcoCore.TcoMessenger(THIS^);
    {attribute 'hide'}
    _progress : INT := 0;
    {attribute 'hide'}
    _infoTimer : TON;
    {attribute 'hide'}
    _errorTimer : TON;
    {attribute 'hide'}
    _timer : TON;
    {attribute 'hide'}
    _varInfo : __SYSTEM.VAR_INFO;
    {attribute 'hide'}
    _sb : TcoCore.StringBuilder;
    {attribute 'hide'}
    _blink : TcoUtilities.TcoBlinker(THIS^);
END_VAR

METHOD CallTimers
VAR_INPUT
    inValue : BOOL;
END_VAR
IF __ISVALIDREF(inoConfig) AND THIS^.inoConfig.ErrorTime <> T#0S OR NOT inValue THEN
    _errorTimer(IN := inValue, PT := THIS^.inoConfig.ErrorTime);
END_IF;

IF __ISVALIDREF(inoConfig) AND THIS^.inoConfig.InfoTime <> T#0S OR NOT inValue THEN
    _infoTimer(IN := inValue, PT := THIS^.inoConfig.InfoTime);
END_IF;
END_METHOD

(*~
    <docu>
        <summary>
            Restores this instance to the Ready state. Can be called explicitly or from within one of the restore mechanisms.
            <para>
                See also <see cref="PlcDocu.TcoCore.TcoTask.AutoRestorable()"/>
            </para>
        </summary>
    </docu>
~*)
METHOD Restore : ITcoRestorable
SUPER^.Restore();
_progress := 0;
_timer(In := FALSE);
CallTimers(FALSE);
Messenger.UnPin();
_errorMessage.UnPin();
END_METHOD

END_FUNCTION_BLOCK

// ---- POUs/Prototypes/RoboticsTasks/Starts/StartMotorsAndProgramTask.TcPOU
FUNCTION_BLOCK StartMotorsAndProgramTask EXTENDS TcoUrRoboticsTask

IF Execute() THEN
    _blink(inOnTime := T#500MS, inOffTime := T#500MS);

    IF _progress = 0 THEN
        IF NOT __ISVALIDREF(inoControl) THEN
            _varInfo := __VARINFO(inoControl);
            Messenger.Programming(_sb.Clear().Append('<#Invalid reference: #>').Append(_varInfo.Symbol).ToString()).Pin();
        ELSIF NOT __ISVALIDREF(inoConfig) THEN
            _varInfo := __VARINFO(inoConfig);
            Messenger.Programming(_sb.Clear().Append('<#Invalid reference: #>').Append(_varInfo.Symbol).ToString()).Pin();
        ELSIF NOT __ISVALIDREF(inoStatus) THEN
            _varInfo := __VARINFO(inoStatus);
            Messenger.Programming(_sb.Clear().Append('<#Invalid reference: #>').Append(_varInfo.Symbol).ToString()).Pin();
        ELSE
            _progress := _progress + 1;
        END_IF
    END_IF

    IF _progress = 1 THEN
        THIS^.Messenger.OnCondition(_infoTimer.Q AND NOT inoStatus.State.Inputs.Safety.NO_IsNormalMode)
            .Warning(_sb.Clear().Append('<# Waiting to Normal Mode. #>').ToString());

        THIS^.Messenger.OnCondition(_infoTimer.Q AND NOT inoStatus.State.Inputs.Safety.RD_IsReducedMode)
            .Warning(_sb.Clear().Append('<# Waiting to Reduced Mode. #>').ToString());

        IF inoStatus.State.Inputs.Safety.NO_IsNormalMode OR inoStatus.State.Inputs.Safety.RD_IsReducedMode THEN
            _progress := _progress + 1;
        END_IF
    END_IF;

    IF _progress = 2 THEN
        Messenger.Warning('<#Robot has error Reset#>');

        IF NOT inoStatus.State.Inputs.Safety.FT_IsFault THEN
            _progress := _progress + 1;
        END_IF
    END_IF;

    IF _progress = 3 THEN
        Messenger.Debug('<#Robot Emergency Stop Reset#>');
        _varInfo := __VARINFO(inoStatus.State.Inputs.Safety.ES_IsEmergencyStopped);

        THIS^.Messenger.OnCondition(_infoTimer.Q AND NOT inoStatus.State.Inputs.Safety.ES_IsEmergencyStopped)
            .Warning(_sb.Clear().Append('<# Waiting for signal: #>').Append(_varInfo.Symbol).ToString());

        _varInfo := __VARINFO(inoStatus.State.Inputs.Safety.PS_IsProtectiveStopped);

        THIS^.Messenger.OnCondition(_infoTimer.Q AND NOT inoStatus.State.Inputs.Safety.PS_IsProtectiveStopped)
            .Warning(_sb.Clear().Append('<# Waiting for signal: #>').Append(_varInfo.Symbol).ToString());

        _varInfo := __VARINFO(inoStatus.State.Inputs.Safety.SS_IsSafeguardStopped);

        THIS^.Messenger.OnCondition(_infoTimer.Q AND NOT inoStatus.State.Inputs.Safety.SS_IsSafeguardStopped)
            .Warning(_sb.Clear().Append('<# Waiting for signal: #>').Append(_varInfo.Symbol).ToString());

        _varInfo := __VARINFO(inoStatus.State.Inputs.Safety.RC_IsRecoveryMode);

        THIS^.Messenger.OnCondition(_infoTimer.Q AND NOT inoStatus.State.Inputs.Safety.RC_IsRecoveryMode)
            .Warning(_sb.Clear().Append('<# Waiting for signal: #>').Append(_varInfo.Symbol).ToString());

        _varInfo := __VARINFO(inoStatus.State.Inputs.Safety.ST_IsStoppedDueSafety);

        THIS^.Messenger.OnCondition(_infoTimer.Q AND NOT inoStatus.State.Inputs.Safety.ES_IsEmergencyStopped)
            .Warning(_sb.Clear().Append('<# Waiting for signal: #>').Append(_varInfo.Symbol).ToString());

        _varInfo := __VARINFO(inoStatus.State.Inputs.Safety.VL_IsViolation);

        THIS^.Messenger.OnCondition(_infoTimer.Q AND NOT inoStatus.State.Inputs.Safety.VL_IsViolation)
            .Warning(_sb.Clear().Append('<# Waiting for signal: #>').Append(_varInfo.Symbol).ToString());

        IF NOT inoStatus.State.Inputs.Safety.ES_IsEmergencyStopped AND
            NOT inoStatus.State.Inputs.Safety.PS_IsProtectiveStopped AND
            NOT inoStatus.State.Inputs.Safety.SS_IsSafeguardStopped AND
            NOT inoStatus.State.Inputs.Safety.RC_IsRecoveryMode AND
            NOT inoStatus.State.Inputs.Safety.ST_IsStoppedDueSafety AND
            NOT inoStatus.State.Inputs.Safety.VL_IsViolation THEN
            _progress := _progress + 1;
        END_IF
    END_IF;

    IF _progress = 4 THEN
        IF inoStatus.State.Inputs.Safety.FT_IsFault THEN
            _progress := 1;
        END_IF

        Messenger.Debug('<#Robot Power on#>');
        _varInfo := __VARINFO(inoStatus.State.Inputs.Robot.PW_IsPowerOn);

        THIS^.Messenger.OnCondition(_infoTimer.Q AND NOT inoStatus.State.Inputs.Robot.PW_IsPowerOn)
            .Warning(_sb.Clear().Append('<# Waiting for signal: #>').Append(_varInfo.Symbol).ToString());

        _varInfo := __VARINFO(inoStatus.State.Inputs.Safety.FT_IsFault);

        THIS^.Messenger.OnCondition(_infoTimer.Q AND NOT inoStatus.State.Inputs.Safety.FT_IsFault)
            .Warning(_sb.Clear().Append('<# Waiting for signal: #>').Append(_varInfo.Symbol).ToString());

        inoControl.MotorOn := _blink.outQ;

        IF inoStatus.State.Inputs.Robot.PW_IsPowerOn AND NOT inoStatus.State.Inputs.Safety.FT_IsFault THEN
            inoControl.MotorOn := FALSE;
            _progress := _progress + 1;
        END_IF
    END_IF;

    IF _progress = 5 THEN
        IF inoStatus.State.Inputs.Safety.FT_IsFault THEN
            _progress := 1;
        END_IF

        inoControl.Start := _blink.outQ;

        THIS^.Messenger.OnCondition(_infoTimer.Q AND NOT inoStatus.State.Inputs.Robot.PR_IsProgramRunning)
            .Warning(_sb.Clear().Append('<#Waiting to program running! #>').ToString());

        IF inoStatus.State.Inputs.Robot.PR_IsProgramRunning AND NOT inoStatus.State.Inputs.Safety.FT_IsFault THEN
            inoControl.Start := FALSE;
        END_IF
    END_IF;

    DoneWhen(inoStatus.State.Inputs.Robot.PR_IsProgramRunning AND
            inoStatus.State.Inputs.Robot.PW_IsPowerOn AND
            NOT inoStatus.State.Inputs.Safety.FT_IsFault);

    CallTimers(TRUE);
    THIS^.ThrowWhen(_errorTimer.Q);
END_IF

IF THIS^.Error AND NOT _errorMessage.Pinned THEN
    THIS^.Restore();
END_IF

(*~
    <docu>
        <summary>
            Executes when task is aborted.
        </summary>
    </docu>
~*)
METHOD PROTECTED OnAbort
IF __ISVALIDREF(inoStatus) THEN
    THIS^.inoStatus.ActionDescription := '<#Start motors and program was aborted.#>';
END_IF;
END_METHOD

(*~
    <docu>
        <summary>
            Executes when task reaches the ```Done``` state .
        </summary>
    </docu>
~*)
METHOD PROTECTED OnDone
IF __ISVALIDREF(inoStatus) THEN
    THIS^.inoStatus.ActionDescription := '<#Start motors and program finished successfully.#>';
END_IF;

_progress := 0;
END_METHOD

METHOD PROTECTED OnError
VAR
    description : STRING;
END_VAR
description := '<#Start motors and program finished with error.#>';

IF __ISVALIDREF(inoStatus) THEN
    THIS^.inoStatus.ActionDescription := description;
END_IF;

THIS^._errorMessage.Error(_sb.Clear().Append(description).Append(' To restore acknowledge this alarm.').ToString()).Pin();
END_METHOD

METHOD PROTECTED OnStart
IF __ISVALIDREF(inoStatus) THEN
    THIS^.inoStatus.ActionDescription := '<#Start motors and program started.#>';
END_IF;

CallTimers(FALSE);
END_METHOD

(*~
    <docu>
        <summary>
            Restores this instance to the Ready state. Can be called explicitly or from within one of the restore mechanisms.
            <para>
                See also <see cref="PlcDocu.TcoCore.TcoTask.AutoRestorable()"/>
            </para>
        </summary>
    </docu>
~*)
METHOD Restore : ITcoRestorable
SUPER^.Restore();
END_METHOD

END_FUNCTION_BLOCK

// ---- POUs/Prototypes/RoboticsTasks/Starts/StartProgramTask.TcPOU
FUNCTION_BLOCK StartProgramTask EXTENDS TcoUrRoboticsTask
VAR
    _stopType : TcoAbstractions.eTcoRoboticsStopType;
END_VAR

IF Execute() THEN
    _blink(inOnTime := T#500MS, inOffTime := T#500MS);

    IF _progress = 0 THEN
        IF NOT __ISVALIDREF(inoControl) THEN
            _varInfo := __VARINFO(inoControl);
            Messenger.Programming(_sb.Clear().Append('<#Invalid reference: #>').Append(_varInfo.Symbol).ToString()).Pin();
        ELSIF NOT __ISVALIDREF(inoConfig) THEN
            _varInfo := __VARINFO(inoConfig);
            Messenger.Programming(_sb.Clear().Append('<#Invalid reference: #>').Append(_varInfo.Symbol).ToString()).Pin();
        ELSIF NOT __ISVALIDREF(inoStatus) THEN
            _varInfo := __VARINFO(inoStatus);
            Messenger.Programming(_sb.Clear().Append('<#Invalid reference: #>').Append(_varInfo.Symbol).ToString()).Pin();
        ELSE
            _progress := _progress + 1;
        END_IF
    END_IF

    IF _progress = 1 THEN
        THIS^.Messenger.OnCondition(_infoTimer.Q AND NOT inoStatus.State.Inputs.Safety.NO_IsNormalMode)
            .Warning(_sb.Clear().Append('<# Waiting to Normal Mode. #>').ToString());

        THIS^.Messenger.OnCondition(_infoTimer.Q AND NOT inoStatus.State.Inputs.Safety.RD_IsReducedMode)
            .Warning(_sb.Clear().Append('<# Waiting to Reduced Mode. #>').ToString());

        IF inoStatus.State.Inputs.Safety.NO_IsNormalMode OR inoStatus.State.Inputs.Safety.RD_IsReducedMode THEN
            _progress := _progress + 1;
        END_IF
    END_IF;

    IF _progress = 2 THEN
        inoControl.Start := _blink.outQ;

        THIS^.Messenger.OnCondition(_infoTimer.Q AND NOT inoStatus.State.Inputs.Robot.PR_IsProgramRunning)
            .Warning(_sb.Clear().Append('<#Waiting to program running! #>').ToString());

        IF inoStatus.State.Inputs.Robot.PR_IsProgramRunning THEN
            inoControl.Start := FALSE;
            _progress := 0;
        END_IF
    END_IF

    DoneWhen(inoStatus.State.Inputs.Robot.PR_IsProgramRunning);
    CallTimers(TRUE);
    THIS^.ThrowWhen(_errorTimer.Q);
END_IF

IF THIS^.Error AND NOT _errorMessage.Pinned THEN
    THIS^.Restore();
END_IF

METHOD INTERNAL InvokeWithParams : ITcoTaskStatus
VAR_INPUT
    inStopType : eTcoRoboticsStopType;
END_VAR
_stopType := inStopType;
InvokeWithParams := THIS^.Invoke();
END_METHOD

(*~
    <docu>
        <summary>
            Executes when task is aborted.
        </summary>
    </docu>
~*)
METHOD PROTECTED OnAbort
IF __ISVALIDREF(inoStatus) THEN
    THIS^.inoStatus.ActionDescription := '<#Stop program was aborted, while not yet completed!#>';
END_IF;
END_METHOD

(*~
    <docu>
        <summary>
            Executes when task reaches the ```Done``` state .
        </summary>
    </docu>
~*)
METHOD PROTECTED OnDone
IF __ISVALIDREF(inoStatus) THEN
    THIS^.inoStatus.ActionDescription := '<#Stop program was completed successfully.#>';
END_IF;

_progress := 0;
END_METHOD

(*~
    <docu>
        <summary>
            Executes when task reaches the ```Error``` state.
                </summary>
    </docu>
~*)
METHOD PROTECTED OnError
VAR
    description : STRING;
END_VAR
THIS^.inoStatus.ActionDescription := '<#Stopping program with error.#>';

IF __ISVALIDREF(inoStatus) THEN
    THIS^.inoStatus.ActionDescription := description;
END_IF;

THIS^._errorMessage.Error(_sb.Clear().Append(description).Append(' To restore acknowledge this alarm.').ToString()).Pin();
END_METHOD

METHOD PROTECTED OnStart
IF __ISVALIDREF(inoStatus) THEN
    THIS^.inoStatus.ActionDescription := '<#Stopping program started.#>';
END_IF;

CallTimers(FALSE);
END_METHOD

(*~
    <docu>
        <summary>
            Restores this instance to the Ready state. Can be called explicitly or from within one of the restore mechanisms.
            <para>
                See also <see cref="PlcDocu.TcoCore.TcoTask.AutoRestorable()"/>
            </para>
        </summary>
    </docu>
~*)
METHOD Restore : ITcoRestorable
SUPER^.Restore();
END_METHOD

END_FUNCTION_BLOCK

// ---- POUs/Prototypes/RoboticsTasks/Starts/StartMotorsTask.TcPOU
FUNCTION_BLOCK StartMotorsTask EXTENDS TcoUrRoboticsTask

IF Execute() THEN
    _blink(inOnTime := T#500MS, inOffTime := T#500MS);

    IF _progress = 0 THEN
        IF NOT __ISVALIDREF(inoControl) THEN
            _varInfo := __VARINFO(inoControl);
            Messenger.Programming(_sb.Clear().Append('<#Invalid reference: #>').Append(_varInfo.Symbol).ToString()).Pin();
        ELSIF NOT __ISVALIDREF(inoConfig) THEN
            _varInfo := __VARINFO(inoConfig);
            Messenger.Programming(_sb.Clear().Append('<#Invalid reference: #>').Append(_varInfo.Symbol).ToString()).Pin();
        ELSIF NOT __ISVALIDREF(inoStatus) THEN
            _varInfo := __VARINFO(inoStatus);
            Messenger.Programming(_sb.Clear().Append('<#Invalid reference: #>').Append(_varInfo.Symbol).ToString()).Pin();
        ELSE
            _progress := _progress + 1;
        END_IF
    END_IF

    IF _progress = 1 THEN
        THIS^.Messenger.OnCondition(_infoTimer.Q AND NOT inoStatus.State.Inputs.Safety.NO_IsNormalMode)
            .Warning(_sb.Clear().Append('<# Waiting to Normal Mode. #>').ToString());

        THIS^.Messenger.OnCondition(_infoTimer.Q AND NOT inoStatus.State.Inputs.Safety.RD_IsReducedMode)
            .Warning(_sb.Clear().Append('<# Waiting to Reduced Mode. #>').ToString());

        IF inoStatus.State.Inputs.Safety.NO_IsNormalMode OR inoStatus.State.Inputs.Safety.RD_IsReducedMode THEN
            _progress := _progress + 1;
        END_IF
    END_IF;

    IF _progress = 2 THEN
        Messenger.Warning('<#Robot has error Reset#>');

        IF NOT inoStatus.State.Inputs.Safety.FT_IsFault THEN
            _progress := _progress + 1;
        END_IF
    END_IF;

    IF _progress = 3 THEN
        Messenger.Debug('<#Robot Emergency Stop Reset#>');
        _varInfo := __VARINFO(inoStatus.State.Inputs.Safety.ES_IsEmergencyStopped);

        THIS^.Messenger.OnCondition(_infoTimer.Q AND NOT inoStatus.State.Inputs.Safety.ES_IsEmergencyStopped)
            .Warning(_sb.Clear().Append('<# Waiting for signal: #>').Append(_varInfo.Symbol).ToString());

        _varInfo := __VARINFO(inoStatus.State.Inputs.Safety.PS_IsProtectiveStopped);

        THIS^.Messenger.OnCondition(_infoTimer.Q AND NOT inoStatus.State.Inputs.Safety.PS_IsProtectiveStopped)
            .Warning(_sb.Clear().Append('<# Waiting for signal: #>').Append(_varInfo.Symbol).ToString());

        _varInfo := __VARINFO(inoStatus.State.Inputs.Safety.SS_IsSafeguardStopped);

        THIS^.Messenger.OnCondition(_infoTimer.Q AND NOT inoStatus.State.Inputs.Safety.SS_IsSafeguardStopped)
            .Warning(_sb.Clear().Append('<# Waiting for signal: #>').Append(_varInfo.Symbol).ToString());

        _varInfo := __VARINFO(inoStatus.State.Inputs.Safety.RC_IsRecoveryMode);

        THIS^.Messenger.OnCondition(_infoTimer.Q AND NOT inoStatus.State.Inputs.Safety.RC_IsRecoveryMode)
            .Warning(_sb.Clear().Append('<# Waiting for signal: #>').Append(_varInfo.Symbol).ToString());

        _varInfo := __VARINFO(inoStatus.State.Inputs.Safety.ST_IsStoppedDueSafety);

        THIS^.Messenger.OnCondition(_infoTimer.Q AND NOT inoStatus.State.Inputs.Safety.ES_IsEmergencyStopped)
            .Warning(_sb.Clear().Append('<# Waiting for signal: #>').Append(_varInfo.Symbol).ToString());

        _varInfo := __VARINFO(inoStatus.State.Inputs.Safety.VL_IsViolation);

        THIS^.Messenger.OnCondition(_infoTimer.Q AND NOT inoStatus.State.Inputs.Safety.VL_IsViolation)
            .Warning(_sb.Clear().Append('<# Waiting for signal: #>').Append(_varInfo.Symbol).ToString());

        //inoControl.ResetEmgStop := inoStatus.State.EmgStop AND _blink.outQ;
        IF NOT inoStatus.State.Inputs.Safety.ES_IsEmergencyStopped AND
            NOT inoStatus.State.Inputs.Safety.PS_IsProtectiveStopped AND
            NOT inoStatus.State.Inputs.Safety.SS_IsSafeguardStopped AND
            NOT inoStatus.State.Inputs.Safety.RC_IsRecoveryMode AND
            NOT inoStatus.State.Inputs.Safety.ST_IsStoppedDueSafety AND
            NOT inoStatus.State.Inputs.Safety.VL_IsViolation THEN
            //inoControl.ResetEmgStop:=FALSE;
            _progress := _progress + 1;
        END_IF
    END_IF;

    IF _progress = 4 THEN
        IF inoStatus.State.Inputs.Safety.FT_IsFault THEN
            _progress := 1;
        END_IF

        Messenger.Debug('<#Robot Power on#>');
        _varInfo := __VARINFO(inoStatus.State.Inputs.Robot.PW_IsPowerOn);

        THIS^.Messenger.OnCondition(_infoTimer.Q AND NOT inoStatus.State.Inputs.Robot.PW_IsPowerOn)
            .Warning(_sb.Clear().Append('<# Waiting for signal: #>').Append(_varInfo.Symbol).ToString());

        _varInfo := __VARINFO(inoStatus.State.Inputs.Safety.FT_IsFault);

        THIS^.Messenger.OnCondition(_infoTimer.Q AND NOT inoStatus.State.Inputs.Safety.FT_IsFault)
            .Warning(_sb.Clear().Append('<# Waiting for signal: #>').Append(_varInfo.Symbol).ToString());

        inoControl.MotorOn := _blink.outQ;

        IF inoStatus.State.Inputs.Robot.PW_IsPowerOn AND
            NOT inoStatus.State.Inputs.Safety.FT_IsFault AND
            inoStatus.State.Inputs.Joints.JointMode[0] = 253 AND
            inoStatus.State.Inputs.Joints.JointMode[1] = 253 AND
            inoStatus.State.Inputs.Joints.JointMode[2] = 253 AND
            inoStatus.State.Inputs.Joints.JointMode[3] = 253 AND
            inoStatus.State.Inputs.Joints.JointMode[4] = 253 AND
            inoStatus.State.Inputs.Joints.JointMode[5] = 253 THEN
            inoControl.MotorOn := FALSE;
            _progress := _progress + 1;
        END_IF
    END_IF;

    DoneWhen(inoStatus.State.Inputs.Robot.PW_IsPowerOn AND
            NOT inoStatus.State.Inputs.Safety.FT_IsFault AND
            inoStatus.State.Inputs.Joints.JointMode[0] = 253 AND
            inoStatus.State.Inputs.Joints.JointMode[1] = 253 AND
            inoStatus.State.Inputs.Joints.JointMode[2] = 253 AND
            inoStatus.State.Inputs.Joints.JointMode[3] = 253 AND
            inoStatus.State.Inputs.Joints.JointMode[4] = 253 AND
            inoStatus.State.Inputs.Joints.JointMode[5] = 253);

    CallTimers(TRUE);
    THIS^.ThrowWhen(_errorTimer.Q);
END_IF

IF THIS^.Error AND NOT _errorMessage.Pinned THEN
    THIS^.Restore();
END_IF

(*~
    <docu>
        <summary>
            Executes when task is aborted.
        </summary>
    </docu>
~*)
METHOD PROTECTED OnAbort
IF __ISVALIDREF(inoStatus) THEN
    THIS^.inoStatus.ActionDescription := '<#Start motors  was aborted.#>';
END_IF;
END_METHOD

(*~
    <docu>
        <summary>
            Executes when task reaches the ```Done``` state .
        </summary>
    </docu>
~*)
METHOD PROTECTED OnDone
IF __ISVALIDREF(inoStatus) THEN
    THIS^.inoStatus.ActionDescription := '<#Start motors  finished successfully.#>';
END_IF;

_progress := 0;
END_METHOD

METHOD PROTECTED OnError
VAR
    description : STRING;
END_VAR
description := '<#Start motors finished with error.#>';

IF __ISVALIDREF(inoStatus) THEN
    THIS^.inoStatus.ActionDescription := description;
END_IF;

THIS^._errorMessage.Error(_sb.Clear().Append(description).Append(' To restore acknowledge this alarm.').ToString()).Pin();
END_METHOD

METHOD PROTECTED OnStart
IF __ISVALIDREF(inoStatus) THEN
    THIS^.inoStatus.ActionDescription := '<#Start motors started.#>';
END_IF;

CallTimers(FALSE);
END_METHOD

(*~
    <docu>
        <summary>
            Restores this instance to the Ready state. Can be called explicitly or from within one of the restore mechanisms.
            <para>
                See also <see cref="PlcDocu.TcoCore.TcoTask.AutoRestorable()"/>
            </para>
        </summary>
    </docu>
~*)
METHOD Restore : ITcoRestorable
SUPER^.Restore();
END_METHOD

END_FUNCTION_BLOCK

// ---- POUs/Prototypes/RoboticsTasks/Starts/StartMovementsTask.TcPOU
FUNCTION_BLOCK StartMovementsTask EXTENDS TcoUrRoboticsTask
VAR
    _moveParams : TcoAbstractions.TcoRoboticsMovementsParams;
END_VAR

IF Execute() THEN
    IF _progress = 0 THEN
        IF NOT __ISVALIDREF(inoControl) THEN
            _varInfo := __VARINFO(inoControl);
            Messenger.Programming(_sb.Clear().Append('<#Invalid reference: #>').Append(_varInfo.Symbol).ToString()).Pin();
        ELSIF NOT __ISVALIDREF(inoConfig) THEN
            _varInfo := __VARINFO(inoConfig);
            Messenger.Programming(_sb.Clear().Append('<#Invalid reference: #>').Append(_varInfo.Symbol).ToString()).Pin();
        ELSIF NOT __ISVALIDREF(inoStatus) THEN
            _varInfo := __VARINFO(inoStatus);
            Messenger.Programming(_sb.Clear().Append('<#Invalid reference: #>').Append(_varInfo.Symbol).ToString()).Pin();
        ELSE
            _progress := _progress + 1;
        END_IF
    END_IF

    IF _progress = 1 THEN
        THIS^.Messenger.OnCondition(_infoTimer.Q AND NOT inoStatus.State.Inputs.Robot.PR_IsProgramRunning)
            .Warning(_sb.Clear().Append('<#Waiting to program running! #>').ToString());

        _varInfo := __VARINFO(inoStatus.State.Inputs.Robot.PW_IsPowerOn);

        THIS^.Messenger.OnCondition(_infoTimer.Q AND NOT inoStatus.State.Inputs.Robot.PW_IsPowerOn)
            .Warning(_sb.Clear().Append('<#Waiting for motors are On! #>').Append(_varInfo.Symbol).ToString());

        _varInfo := __VARINFO(inoStatus.State.Inputs.Safety.FT_IsFault);

        THIS^.Messenger.OnCondition(_infoTimer.Q AND inoStatus.State.Inputs.Safety.FT_IsFault)
            .Warning(_sb.Clear().Append('<#Waiting for system is without errors! #>').Append(_varInfo.Symbol).ToString());

        IF inoStatus.State.Inputs.Robot.PR_IsProgramRunning AND
            inoStatus.State.Inputs.Robot.PW_IsPowerOn AND
            NOT inoStatus.State.Inputs.Safety.FT_IsFault THEN
            _progress := _progress + 1;
        END_IF
    END_IF;

    IF _progress = 2 THEN
        inoControl.GlobalSpeed := _moveParams.GlobalSpeed;
        inoControl.ToolNo := _moveParams.ToolNo;
        inoControl.WorkobjectNo := _moveParams.WorkobjectNo;
        inoControl.PointNo := _moveParams.PointNo;
        inoControl.UserSpecSpeed1 := _moveParams.UserSpecSpeed1;
        inoControl.UserSpecSpeed2 := _moveParams.UserSpecSpeed2;
        inoControl.Coordinates := _moveParams.Coordinates;
        inoControl.ActionNo := 254;

        IF inoControl.ActionNo = inoStatus.State.ActionNo THEN
            _progress := _progress + 1;
        END_IF
    END_IF;

    IF _progress = 3 THEN
        IF inoStatus.State.GlobalSpeed = _moveParams.GlobalSpeed AND
            inoStatus.State.ToolNo = _moveParams.ToolNo AND
            inoStatus.State.WorkobjectNo = _moveParams.WorkobjectNo AND
            inoStatus.State.PointNo = _moveParams.PointNo AND
            inoStatus.State.UserSpecSpeed1 = _moveParams.UserSpecSpeed1 AND
            inoStatus.State.UserSpecSpeed2 = _moveParams.UserSpecSpeed2 AND
            TcoAbstractions.CoordinatesAreEqual(inoStatus.State.Coordinates,
                _moveParams.Coordinates,
                0.01,
                0.01,
                0.01,
                0.01,
                0.01,
                0.01) THEN
            inoControl.ActionNo := 255;
            _progress := _progress + 1;
        END_IF
    END_IF;

    IF _progress = 4 THEN
        IF inoControl.ActionNo = inoStatus.State.ActionNo THEN
            _progress := _progress + 1;
        END_IF
    END_IF;

    IF _progress = 5 THEN
        Messenger.Info(CONCAT('<#Moving to position ID#>: ', INT_TO_STRING(_moveParams.ActionNo)));
        inoControl.ActionNo := _moveParams.ActionNo;

